// TIA Portal V17 export
// export: Created 2025-03-10T12:16:33.8598493Z, ExportSetting WithDefaults, DisplayName Totally Integrated Automation Portal, DisplayVersion V17 Update 8, DisplayName TIA Portal Openness, DisplayVersion V17 Update 8, DisplayName TIA Portal Version Control Interface, DisplayVersion V17, DisplayName SINAMICS Startdrive Advanced, DisplayVersion V17 SP2, DisplayName SINAMICS Startdrive G110M, G120, G120C, G120D, G120P, G115D, DisplayVersion V17 SP2, DisplayName SINAMICS Startdrive G130, G150, S120, S150, SINAMICS MV, S210, DisplayVersion V17 SP2, DisplayName STEP 7 Professional, DisplayVersion V17 Update 8, DisplayName SINUMERIK ONE STEP 7 Toolbox, DisplayVersion V17 Update 12, DisplayName SINUMERIK 840D sl STEP 7 Toolbox, DisplayVersion V17 Update 12, DisplayName STEP 7 Safety, DisplayVersion V17 Update 6, DisplayName WinCC Advanced, DisplayVersion V17 Update 8
FUNCTION_BLOCK "FB1452_AUXILIARY_COOLING_SYSTEM"   // FB1452, LAD
{ S7_Optimized_Access := 'FALSE' }
AUTHOR : ETXETAR
VERSION : 1.0
// stored: AutoNumber false, IsIECCheckEnabled false, SetENOAutomatically false, UDAEnableTagReadback false
   VAR_INPUT
      OPTIONS_0 : Byte := 2#0000_0000;   // OPTIONS 0
      OPTIONS_1 : Byte := 2#0000_0000;   // OPTIONS 1
      CIRCUIT_BREAKER_INPUT : Bool;   // CIRCUIT BREAKER INPUT
      CONTACTOR_FEEDBACK : Bool;   // CONTACTOR FEEDBACK INPUT
      LOW_LEVEL_ALM : Bool;   // UNIT 01 LOW LEVEL ALARM
      OVERTEMPERATURE_ALM : Bool;   // UNIT 01 OVERTEMPERATURE ALARM
      U01_FLOW_ACTUAL_RAW_VALUE : Int;   // UNIT 01 FLOW ACTUAL RAW VALUE
      U01_TEMP_ACTUAL_RAW_VALUE : Int;   // UNIT 01 TEMPURATURE ACTUAL RAW VALUE
      U02_FLOW_ACTUAL_RAW_VALUE : Int;   // UNIT 02 FLOW ACTUAL RAW VALUE
      U02_TEMP_ACTUAL_RAW_VALUE : Int;   // UNIT 02 TEMPURATURE ACTUAL RAW VALUE
      HMI_REQ_LINE : Bool;   // HMI REQUEST LINE
   END_VAR
   VAR_OUTPUT
      U01_U02_BREAKER_TRIPPED_ALARM : Bool;   // UNIT 01 & UNIT 02 CIRCUIT BREAKER TRIPPED ALARM
      U01_U02_CONTACTOR_FEEDBACK_ALARM : Bool;   // UNIT 01 & UNIT 02 CONTACTOR FEEDBACK ALARM
      U01_U02_LOW_LEVEL_INPUT_ALARM : Bool;   // UNIT 01 & UNIT 02 LOW LEVEL INPUT ALARM
      U01_U02_OVERTEMPERATURE_INPUT_ALARM : Bool;   // UNIT 01 & UNIT 02 OVERTEMPERATURE INPUT ALARM
      U01_FLOW_FEEDBACK_ALARM : Bool;   // UNIT 01 FLOW FEEDBACK ALARM
      U01_FLOW_HIGH_LIMIT_ALARM : Bool;   // UNIT 01 FLOW HIGH LIMIT ALARM
      U01_FLOW_HIGH_LIMIT_WARNING : Bool;   // UNIT 01 FLOW HIGH LIMIT WARNING
      U01_FLOW_LOW_LIMIT_ALARM : Bool;   // UNIT 01 FLOW LOW LIMIT ALARM
      U01_FLOW_LOW_LIMIT_WARNING : Bool;   // UNIT 01 FLOW LOW LIMIT WARNING
      U01_TEMP_HIGH_LIMIT_ALARM : Bool;   // UNIT 01 TEMPERATURE HIGH LIMIT ALARM
      U01_TEMP_HIGH_LIMIT_WARNING : Bool;   // UNIT 01 TEMPERATURE HIGH LIMIT WARNING
      U01_TEMP_LOW_LIMIT_ALARM : Bool;   // UNIT 01 TEMPERATURE LOW LIMIT ALARM
      U01_TEMP_LOW_LIMIT_WARNING : Bool;   // UNIT 01 TEMPERATURE LOW LIMIT WARNING
      U01_FLOW_SETPOINT_ALARM : Bool;   // UNIT 01 FLOW SETPOINT ALARM
      U01_TEMP_SETPOINT_ALARM : Bool;   // UNIT 01 TEMPERATURE SETPOINT ALARM
      U02_FLOW_FEEDBACK_ALARM : Bool;   // UNIT 02 FLOW FEEDBACK ALARM
      U02_FLOW_HIGH_LIMIT_ALARM : Bool;   // UNIT 01 FLOW HIGH LIMIT ALARM
      U02_FLOW_HIGH_LIMIT_WARNING : Bool;   // UNIT 01 FLOW HIGH LIMIT WARNING
      U02_FLOW_LOW_LIMIT_ALARM : Bool;   // UNIT 01 FLOW LOW LIMIT ALARM
      U02_FLOW_LOW_LIMIT_WARNING : Bool;   // UNIT 01 FLOW LOW LIMIT WARNING
      U02_TEMP_HIGH_LIMIT_ALARM : Bool;   // UNIT 01 TEMPERATURE HIGH LIMIT ALARM
      U02_TEMP_HIGH_LIMIT_WARNING : Bool;   // UNIT 01 TEMPERATURE HIGH LIMIT WARNING
      U02_TEMP_LOW_LIMIT_ALARM : Bool;   // UNIT 01 TEMPERATURE LOW LIMIT ALARM
      U02_TEMP_LOW_LIMIT_WARNING : Bool;   // UNIT 01 TEMPERATURE LOW LIMIT WARNING
      U02_FLOW_SETPOINT_ALARM : Bool;   // UNIT 01 FLOW SETPOINT ALARM
      U02_TEMP_SETPOINT_ALARM : Bool;   // UNIT 01 TEMPERATURE SETPOINT ALARM
      HMI_POWER_UP_COND_OFF : Bool;   // HMI POWER UP CONDITIONS OFF
      HMI_POWER_UP_COND_ON : Bool;   // HMI POWER UP CONDITIONS ON
      HMI_POWER_UP_EXECU_LEFT : Bool;   // HMI POWER UP EXECUTABLE LEFT
      HMI_POWER_UP_EXECU_RIGHT : Bool;   // HMI POWER UP EXECUTABLE RIGHT
      MAIN_VALVE : Bool;   // MAIN VALVE OUTPUT
   END_VAR
   VAR DB_SPECIFIC
      SWITCH_ON_GENERAL_CONDITIONS : Bool;   // SWITCH ON GENERAL CONDITIONS
      SWITCH_ON_INITIAL_CONDITIONS : Bool;   // SWITCH ON INITIAL CONDITIONS
      SWITCH_ON_MANUAL_REQUEST : Bool;   // SWITCH ON MANUAL REQUEST
      SWITCH_ON_AUTO_REQUEST : Bool;   // SWITCH ON AUTO REQUEST
      SWITCH_ON_GLOBAL_REQUEST : Bool;   // SWITCH ON GLOBAL REQUEST
      SWITCH_ON_COMMAND : Bool;   // SWITCH ON COMMAND
      SWITCH_ON : Bool;   // SWITCH ON
      IN_SERVICE : Bool;   // IN SERVICE
      SWITCH_OFF_GENERAL_CONDITIONS : Bool;   // SWITCH OFF GENERAL CONDITIONS
      SWITCH_OFF_INITIAL_CONDITIONS : Bool;   // SWITCH OFF INITIAL CONDITIONS
      SWITCH_OFF_MANUAL_REQUEST : Bool;   // SWITCH OFF MANUAL REQUEST
      SWITCH_OFF_AUTO_REQUEST : Bool;   // SWITCH OFF AUTO REQUEST
      SWITCH_OFF_GLOBAL_REQUEST : Bool;   // SWITCH OFF GLOBAL REQUEST
      SWITCH_OFF_COMMAND : Bool;   // SWITCH OFF COMMAND
      SWITCH_OFF : Bool;   // SWITCH OFF
      OUT_OF_SERVICE : Bool;   // OUT OF SERVICE
      MANUAL_REQUEST_HELP : Bool;   // MANUAL REQUEST HELP
      SWITCH_ON_GENERAL_CONDITION_HELP : Bool;   // SWITCH ON GENERAL CONDITION HELP
      SWITCH_ON_INITIAL_CONDITION_HELP : Bool;   // SWITCH ON INITIAL CONDITION HELP
      SWITCH_OFF_GENERAL_CONDITION_HELP : Bool;   // SWITCH OFF GENERAL CONDITION HELP
      SWITCH_OFF_INITIAL_CONDITION_HELP : Bool;   // SWITCH OFF INITIAL CONDITION HELP
      ANY_ACTIVE_ALARM : Bool;   // ANY ACTIVE ALARM
      SEOC_ALARMS : Bool;   // STOP END OF CYCLE ALARMS
      WARNINGS : Bool;   // WARNINGS
      WARNINGS_GONE : Bool;   // WARNINGS GONE
      UNIT_01_FLOW_FEEDBACK_INPUT : Bool;   // UNIT 01 FLOW PRESENT INPUT
      UNIT_02_FLOW_FEEDBACK_INPUT : Bool;   // UNIT 02 FLOW PRESENT INPUT
      TOTAL_FLOW_FEEDBACK_INPUT : Bool;   // TOTAL FLOW PRESENT INPUT
      AUX_COOLING_SENSOR_U01_VALUES { ExternalAccessible := 'False'; ExternalVisible := 'False'; ExternalWritable := 'False'} : "COOLING_SENSOR";
      AUX_COOLING_SENSOR_U02_VALUES { ExternalAccessible := 'False'; ExternalVisible := 'False'; ExternalWritable := 'False'} : "COOLING_SENSOR";
      TIMER_CONVEYOR_CONTACTOR_RELAY_ALARM : TON_TIME;   // PRESSURE TIMER
   END_VAR
   VAR_TEMP
      INPUTS_MASK : Byte;   // INPUT MASK
      O_BYTE_0 : Struct   // OPTIONS BYTE 0
         GEN_CIRCUIT_BREAKER : Bool;   // GENERAL CIRCUIT BREAKER OPTION
         GEN_CONTACTOR_FEEDBACK : Bool;   // GENERAL CONTACTOR FEEDBACK OPTION
         U01_FLOW_SETPOINT_ALARM : Bool;   // UNIT 01 FLOW SETPOINT ALARM
         U01_TEMP_SETPOINT_ALARM : Bool;   // UNIT 01 TEMPERATURE SETPOINT ALARM
         SPARE_2 : Bool;
         SPARE_3 : Bool;
         SPARE_4 : Bool;
         SPARE_5 : Bool;
      END_STRUCT;
      O_BYTE_1 : Struct   // OPTIONS BYTE 1
         FIRST_FEEDBACK_FLOW_TEMP_SENSOR : Bool;   // FIRST FEEDBACK FLOW TEMP SENSOR
         SECOND_FEEDBACK_FLOW_TEMP_SENSOR : Bool;   // SECOND FEEDBACK FLOW TEMP SENSOR
         U02_FLOW_SETPOINT_ALARM : Bool;   // UNIT 02 FLOW SETPOINT ALARM
         U02_TEMP_SETPOINT_ALARM : Bool;   // UNIT 02 TEMPERATURE SETPOINT ALARM
         SPARE_2 : Bool;
         SPARE_3 : Bool;
         SPARE_4 : Bool;
         SPARE_5 : Bool;
      END_STRUCT;
      DB_NUMBER : DInt;   // DB NUMBER FOR ALARM DECODING
      FLOW_AUX : Real;
      TEMPERATURE_AUX : Int;
   END_VAR
   // TIMER_CONVEYOR_CONTACTOR_RELAY_ALARM.PT := T#1M;
   VAR_TEMP   // added for the SCL form of the ladder/FBD networks
      _w1 : Bool;
   END_VAR
BEGIN

NETWORK
TITLE = READ INSTANCE DB
      L     DINO;
      +     10#800000;
      T     #DB_NUMBER;


REGION Network 2: OPTIONS
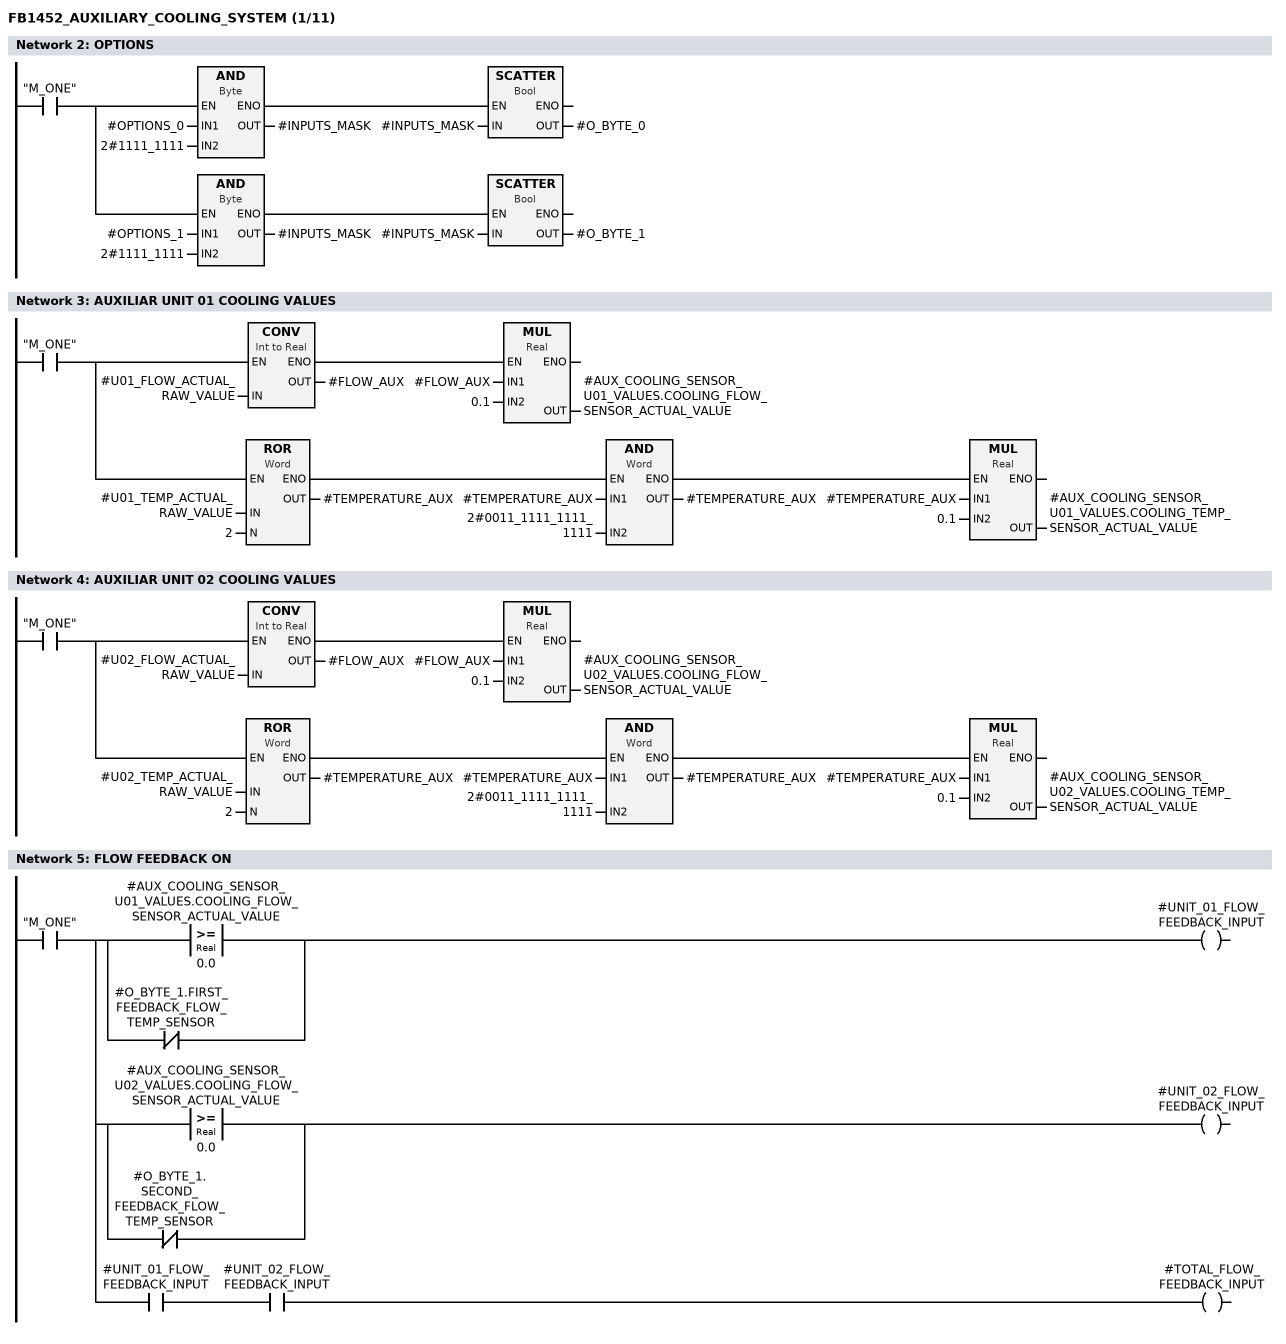
   RUNG wire#powerrail
      Contact( "M_ONE" )
      wire#w1
      { S7_Templates := "SrcType := Byte"; S7_GenerateENO := "TRUE" } And(in1 := #OPTIONS_0, in2 := 2#1111_1111, out => #INPUTS_MASK)
      { S7_Templates := "[dest_type := Bool, src_type := Byte]" } SCATTER(IN := #INPUTS_MASK, OUT => #O_BYTE_0)
   END_RUNG
   RUNG wire#w1
      { S7_Templates := "SrcType := Byte"; S7_GenerateENO := "TRUE" } And(in1 := #OPTIONS_1, in2 := 2#1111_1111, out => #INPUTS_MASK)
      { S7_Templates := "[dest_type := Bool, src_type := Byte]" } SCATTER(IN := #INPUTS_MASK, OUT => #O_BYTE_1)
   END_RUNG
   // the same network as SCL:
   IF "M_ONE" THEN #INPUTS_MASK := #OPTIONS_0 AND 2#1111_1111; END_IF;
   #_w1 := "M_ONE";
   IF #_w1 THEN
       SCATTER(IN := #INPUTS_MASK, OUT => #O_BYTE_0);
       #INPUTS_MASK := #OPTIONS_1 AND 2#1111_1111;
       SCATTER(IN := #INPUTS_MASK, OUT => #O_BYTE_1);
   END_IF;
END_REGION

REGION Network 3: AUXILIAR UNIT 01 COOLING VALUES
   IF "M_ONE" THEN
       #FLOW_AUX := INT_TO_REAL(#U01_FLOW_ACTUAL_RAW_VALUE);
       #AUX_COOLING_SENSOR_U01_VALUES.COOLING_FLOW_SENSOR_ACTUAL_VALUE := #FLOW_AUX * 0.1;
       #TEMPERATURE_AUX := ROR(IN := #U01_TEMP_ACTUAL_RAW_VALUE, N := 2);
       #TEMPERATURE_AUX := #TEMPERATURE_AUX AND 2#0011_1111_1111_1111;
       #AUX_COOLING_SENSOR_U01_VALUES.COOLING_TEMP_SENSOR_ACTUAL_VALUE := #TEMPERATURE_AUX * 0.1;
   END_IF;
END_REGION

REGION Network 4: AUXILIAR UNIT 02 COOLING VALUES
   IF "M_ONE" THEN
       #FLOW_AUX := INT_TO_REAL(#U02_FLOW_ACTUAL_RAW_VALUE);
       #AUX_COOLING_SENSOR_U02_VALUES.COOLING_FLOW_SENSOR_ACTUAL_VALUE := #FLOW_AUX * 0.1;
       #TEMPERATURE_AUX := ROR(IN := #U02_TEMP_ACTUAL_RAW_VALUE, N := 2);
       #TEMPERATURE_AUX := #TEMPERATURE_AUX AND 2#0011_1111_1111_1111;
       #AUX_COOLING_SENSOR_U02_VALUES.COOLING_TEMP_SENSOR_ACTUAL_VALUE := #TEMPERATURE_AUX * 0.1;
   END_IF;
END_REGION

REGION Network 5: FLOW FEEDBACK ON
   RUNG wire#powerrail
      Contact( "M_ONE" )
      wire#w1
      { S7_Templates := "SrcType := Real" } GE_Contact(in1 := #AUX_COOLING_SENSOR_U01_VALUES.COOLING_FLOW_SENSOR_ACTUAL_VALUE, in2 := 0.0)
      wire#w2
      Coil( #UNIT_01_FLOW_FEEDBACK_INPUT )
   END_RUNG
   RUNG wire#w1
      I_Contact( #O_BYTE_1.FIRST_FEEDBACK_FLOW_TEMP_SENSOR )
   END_RUNG wire#w2
   RUNG wire#w1
      { S7_Templates := "SrcType := Real" } GE_Contact(in1 := #AUX_COOLING_SENSOR_U02_VALUES.COOLING_FLOW_SENSOR_ACTUAL_VALUE, in2 := 0.0)
      wire#w3
      Coil( #UNIT_02_FLOW_FEEDBACK_INPUT )
   END_RUNG
   RUNG wire#w1
      I_Contact( #O_BYTE_1.SECOND_FEEDBACK_FLOW_TEMP_SENSOR )
   END_RUNG wire#w3
   RUNG wire#w1
      Contact( #UNIT_01_FLOW_FEEDBACK_INPUT )
      Contact( #UNIT_02_FLOW_FEEDBACK_INPUT )
      Coil( #TOTAL_FLOW_FEEDBACK_INPUT )
   END_RUNG
   // the same network as SCL:
   #UNIT_01_FLOW_FEEDBACK_INPUT := "M_ONE" AND ((#AUX_COOLING_SENSOR_U01_VALUES.COOLING_FLOW_SENSOR_ACTUAL_VALUE >= 0.0) OR NOT #O_BYTE_1.FIRST_FEEDBACK_FLOW_TEMP_SENSOR);
   #UNIT_02_FLOW_FEEDBACK_INPUT := "M_ONE" AND ((#AUX_COOLING_SENSOR_U02_VALUES.COOLING_FLOW_SENSOR_ACTUAL_VALUE >= 0.0) OR NOT #O_BYTE_1.SECOND_FEEDBACK_FLOW_TEMP_SENSOR);
   #TOTAL_FLOW_FEEDBACK_INPUT := "M_ONE" AND #UNIT_01_FLOW_FEEDBACK_INPUT AND #UNIT_02_FLOW_FEEDBACK_INPUT;
END_REGION

REGION Network 6: SWITCH ON GENERAL CONDITIONS
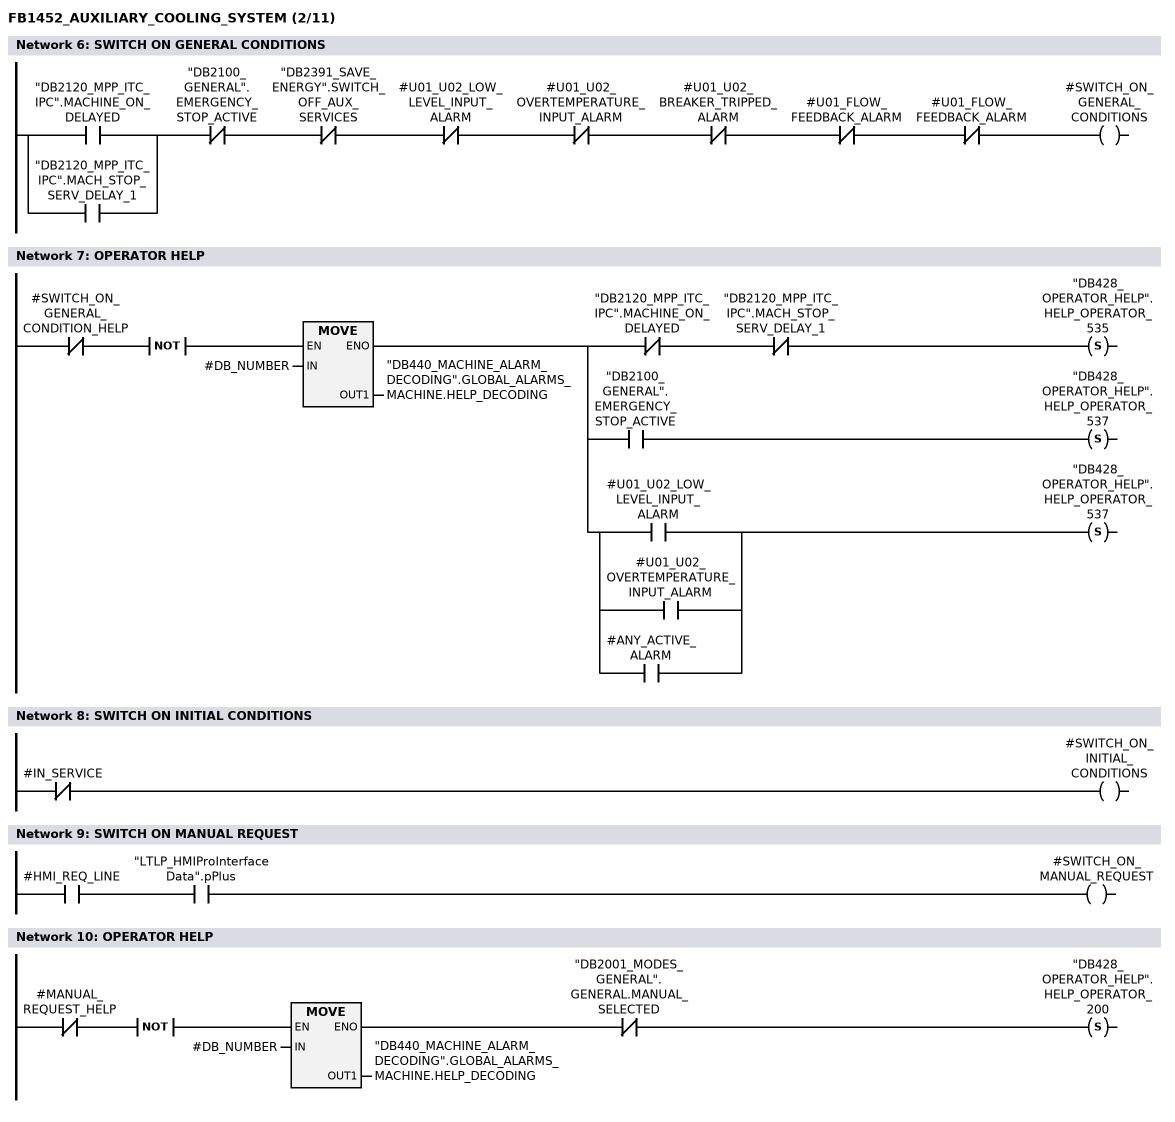
   RUNG wire#powerrail
      Contact( "DB2120_MPP_ITC_IPC".MACHINE_ON_DELAYED )
      wire#w1
      I_Contact( "DB2100_GENERAL".EMERGENCY_STOP_ACTIVE )
      I_Contact( "DB2391_SAVE_ENERGY".SWITCH_OFF_AUX_SERVICES )
      I_Contact( #U01_U02_LOW_LEVEL_INPUT_ALARM )
      I_Contact( #U01_U02_OVERTEMPERATURE_INPUT_ALARM )
      I_Contact( #U01_U02_BREAKER_TRIPPED_ALARM )
      I_Contact( #U01_FLOW_FEEDBACK_ALARM )
      I_Contact( #U01_FLOW_FEEDBACK_ALARM )
      Coil( #SWITCH_ON_GENERAL_CONDITIONS )
   END_RUNG
   RUNG wire#powerrail
      Contact( "DB2120_MPP_ITC_IPC".MACH_STOP_SERV_DELAY_1 )
   END_RUNG wire#w1
   // the same network as SCL:
   #SWITCH_ON_GENERAL_CONDITIONS := ("DB2120_MPP_ITC_IPC".MACHINE_ON_DELAYED OR "DB2120_MPP_ITC_IPC".MACH_STOP_SERV_DELAY_1) AND NOT "DB2100_GENERAL".EMERGENCY_STOP_ACTIVE AND NOT "DB2391_SAVE_ENERGY".SWITCH_OFF_AUX_SERVICES AND NOT #U01_U02_LOW_LEVEL_INPUT_ALARM AND NOT #U01_U02_OVERTEMPERATURE_INPUT_ALARM AND NOT #U01_U02_BREAKER_TRIPPED_ALARM AND NOT #U01_FLOW_FEEDBACK_ALARM AND NOT #U01_FLOW_FEEDBACK_ALARM;
END_REGION

REGION Network 7: OPERATOR HELP
   RUNG wire#powerrail
      I_Contact( #SWITCH_ON_GENERAL_CONDITION_HELP )
      Not()
      { S7_GenerateENO := "TRUE" } Move(in := #DB_NUMBER, out1 => "DB440_MACHINE_ALARM_DECODING".GLOBAL_ALARMS_MACHINE.HELP_DECODING)
      wire#w1
      I_Contact( "DB2120_MPP_ITC_IPC".MACHINE_ON_DELAYED )
      I_Contact( "DB2120_MPP_ITC_IPC".MACH_STOP_SERV_DELAY_1 )
      S_Coil( "DB428_OPERATOR_HELP".HELP_OPERATOR_535 )
   END_RUNG
   RUNG wire#w1
      Contact( "DB2100_GENERAL".EMERGENCY_STOP_ACTIVE )
      S_Coil( "DB428_OPERATOR_HELP".HELP_OPERATOR_537 )
   END_RUNG
   RUNG wire#w1
      Contact( #U01_U02_LOW_LEVEL_INPUT_ALARM )
      wire#w2
      S_Coil( "DB428_OPERATOR_HELP".HELP_OPERATOR_537 )
   END_RUNG
   RUNG wire#w1
      Contact( #U01_U02_OVERTEMPERATURE_INPUT_ALARM )
   END_RUNG wire#w2
   RUNG wire#w1
      Contact( #ANY_ACTIVE_ALARM )
   END_RUNG wire#w2
   // the same network as SCL:
   // ENO of a box is taken as its EN; it also drops when the box reports an error
   #_w1 := NOT (NOT #SWITCH_ON_GENERAL_CONDITION_HELP);
   IF #_w1 THEN "DB440_MACHINE_ALARM_DECODING".GLOBAL_ALARMS_MACHINE.HELP_DECODING := #DB_NUMBER; END_IF;
   IF #_w1 AND NOT "DB2120_MPP_ITC_IPC".MACHINE_ON_DELAYED AND NOT "DB2120_MPP_ITC_IPC".MACH_STOP_SERV_DELAY_1 THEN
       "DB428_OPERATOR_HELP".HELP_OPERATOR_535 := TRUE;
   END_IF;
   IF #_w1 AND "DB2100_GENERAL".EMERGENCY_STOP_ACTIVE THEN
       "DB428_OPERATOR_HELP".HELP_OPERATOR_537 := TRUE;
   END_IF;
   IF #_w1 AND (#U01_U02_LOW_LEVEL_INPUT_ALARM OR #U01_U02_OVERTEMPERATURE_INPUT_ALARM OR #ANY_ACTIVE_ALARM) THEN
       "DB428_OPERATOR_HELP".HELP_OPERATOR_537 := TRUE;
   END_IF;
END_REGION

REGION Network 8: SWITCH ON INITIAL CONDITIONS
   RUNG wire#powerrail
      I_Contact( #IN_SERVICE )
      Coil( #SWITCH_ON_INITIAL_CONDITIONS )
   END_RUNG
   // the same network as SCL:
   #SWITCH_ON_INITIAL_CONDITIONS := NOT #IN_SERVICE;
END_REGION

REGION Network 9: SWITCH ON MANUAL REQUEST
   RUNG wire#powerrail
      Contact( #HMI_REQ_LINE )
      Contact( "LTLP_HMIProInterfaceData".pPlus )
      Coil( #SWITCH_ON_MANUAL_REQUEST )
   END_RUNG
   // the same network as SCL:
   #SWITCH_ON_MANUAL_REQUEST := #HMI_REQ_LINE AND "LTLP_HMIProInterfaceData".pPlus;
END_REGION

REGION Network 10: OPERATOR HELP
   RUNG wire#powerrail
      I_Contact( #MANUAL_REQUEST_HELP )
      Not()
      { S7_GenerateENO := "TRUE" } Move(in := #DB_NUMBER, out1 => "DB440_MACHINE_ALARM_DECODING".GLOBAL_ALARMS_MACHINE.HELP_DECODING)
      I_Contact( "DB2001_MODES_GENERAL".GENERAL.MANUAL_SELECTED )
      S_Coil( "DB428_OPERATOR_HELP".HELP_OPERATOR_200 )
   END_RUNG
   // the same network as SCL:
   // ENO of a box is taken as its EN; it also drops when the box reports an error
   #_w1 := NOT (NOT #MANUAL_REQUEST_HELP);
   IF #_w1 THEN "DB440_MACHINE_ALARM_DECODING".GLOBAL_ALARMS_MACHINE.HELP_DECODING := #DB_NUMBER; END_IF;
   IF #_w1 AND NOT "DB2001_MODES_GENERAL".GENERAL.MANUAL_SELECTED THEN
       "DB428_OPERATOR_HELP".HELP_OPERATOR_200 := TRUE;
   END_IF;
END_REGION

REGION Network 11: SWITCH ON AUTO REQUEST
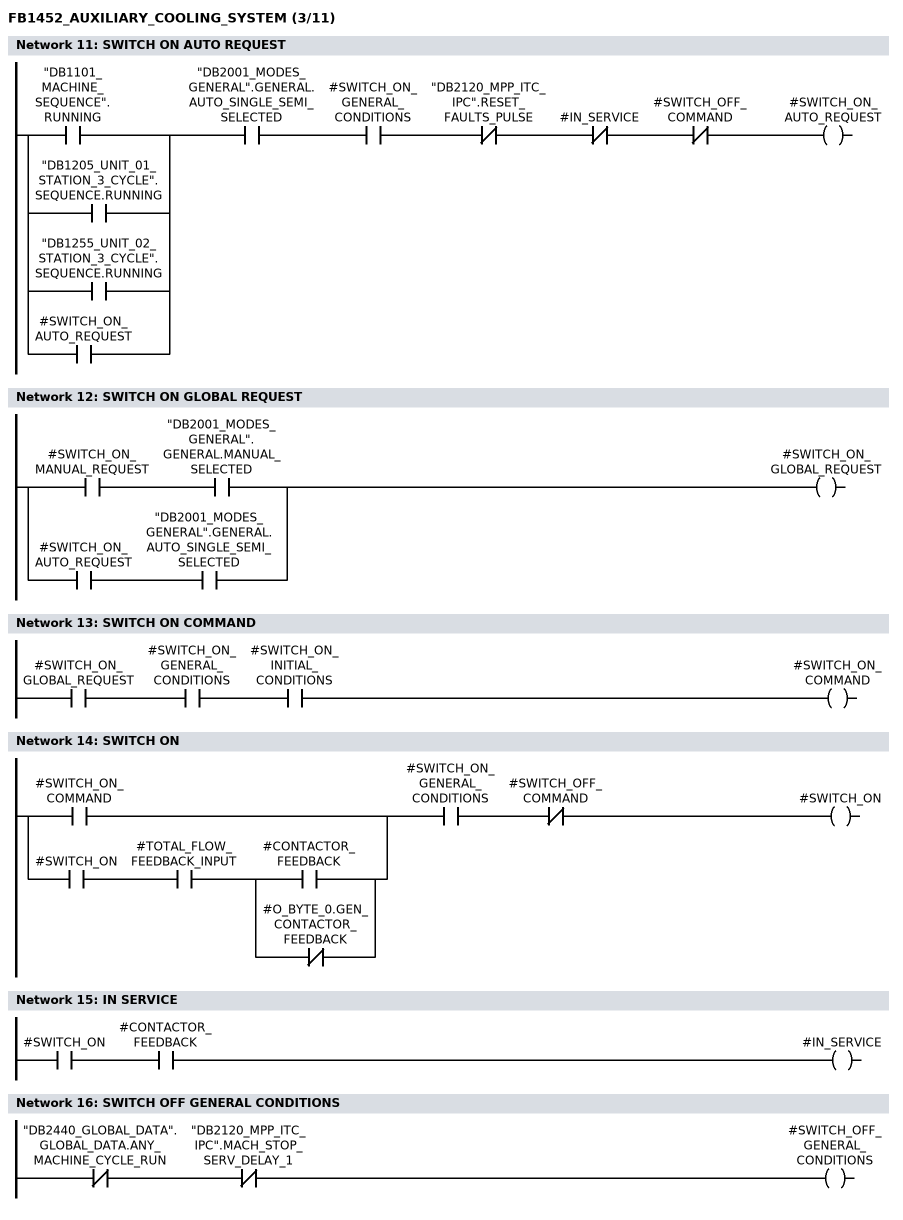
   RUNG wire#powerrail
      Contact( "DB1101_MACHINE_SEQUENCE".RUNNING )
      wire#w1
      Contact( "DB2001_MODES_GENERAL".GENERAL.AUTO_SINGLE_SEMI_SELECTED )
      Contact( #SWITCH_ON_GENERAL_CONDITIONS )
      I_Contact( "DB2120_MPP_ITC_IPC".RESET_FAULTS_PULSE )
      I_Contact( #IN_SERVICE )
      I_Contact( #SWITCH_OFF_COMMAND )
      Coil( #SWITCH_ON_AUTO_REQUEST )
   END_RUNG
   RUNG wire#powerrail
      Contact( "DB1205_UNIT_01_STATION_3_CYCLE".SEQUENCE.RUNNING )
   END_RUNG wire#w1
   RUNG wire#powerrail
      Contact( "DB1255_UNIT_02_STATION_3_CYCLE".SEQUENCE.RUNNING )
   END_RUNG wire#w1
   RUNG wire#powerrail
      Contact( #SWITCH_ON_AUTO_REQUEST )
   END_RUNG wire#w1
   // the same network as SCL:
   #SWITCH_ON_AUTO_REQUEST := ("DB1101_MACHINE_SEQUENCE".RUNNING OR "DB1205_UNIT_01_STATION_3_CYCLE".SEQUENCE.RUNNING OR "DB1255_UNIT_02_STATION_3_CYCLE".SEQUENCE.RUNNING OR #SWITCH_ON_AUTO_REQUEST) AND "DB2001_MODES_GENERAL".GENERAL.AUTO_SINGLE_SEMI_SELECTED AND #SWITCH_ON_GENERAL_CONDITIONS AND NOT "DB2120_MPP_ITC_IPC".RESET_FAULTS_PULSE AND NOT #IN_SERVICE AND NOT #SWITCH_OFF_COMMAND;
END_REGION

REGION Network 12: SWITCH ON GLOBAL REQUEST
   RUNG wire#powerrail
      Contact( #SWITCH_ON_MANUAL_REQUEST )
      Contact( "DB2001_MODES_GENERAL".GENERAL.MANUAL_SELECTED )
      wire#w1
      Coil( #SWITCH_ON_GLOBAL_REQUEST )
   END_RUNG
   RUNG wire#powerrail
      Contact( #SWITCH_ON_AUTO_REQUEST )
      Contact( "DB2001_MODES_GENERAL".GENERAL.AUTO_SINGLE_SEMI_SELECTED )
   END_RUNG wire#w1
   // the same network as SCL:
   #SWITCH_ON_GLOBAL_REQUEST := (#SWITCH_ON_MANUAL_REQUEST AND "DB2001_MODES_GENERAL".GENERAL.MANUAL_SELECTED) OR (#SWITCH_ON_AUTO_REQUEST AND "DB2001_MODES_GENERAL".GENERAL.AUTO_SINGLE_SEMI_SELECTED);
END_REGION

REGION Network 13: SWITCH ON COMMAND
   RUNG wire#powerrail
      Contact( #SWITCH_ON_GLOBAL_REQUEST )
      Contact( #SWITCH_ON_GENERAL_CONDITIONS )
      Contact( #SWITCH_ON_INITIAL_CONDITIONS )
      Coil( #SWITCH_ON_COMMAND )
   END_RUNG
   // the same network as SCL:
   #SWITCH_ON_COMMAND := #SWITCH_ON_GLOBAL_REQUEST AND #SWITCH_ON_GENERAL_CONDITIONS AND #SWITCH_ON_INITIAL_CONDITIONS;
END_REGION

REGION Network 14: SWITCH ON
   RUNG wire#powerrail
      Contact( #SWITCH_ON_COMMAND )
      wire#w1
      Contact( #SWITCH_ON_GENERAL_CONDITIONS )
      I_Contact( #SWITCH_OFF_COMMAND )
      Coil( #SWITCH_ON )
   END_RUNG
   RUNG wire#powerrail
      Contact( #SWITCH_ON )
      Contact( #TOTAL_FLOW_FEEDBACK_INPUT )
      wire#w2
      Contact( #CONTACTOR_FEEDBACK )
   END_RUNG wire#w1
   RUNG wire#w2
      I_Contact( #O_BYTE_0.GEN_CONTACTOR_FEEDBACK )
   END_RUNG wire#w1
   // the same network as SCL:
   #SWITCH_ON := (#SWITCH_ON_COMMAND OR (#SWITCH_ON AND #TOTAL_FLOW_FEEDBACK_INPUT AND (#CONTACTOR_FEEDBACK OR NOT #O_BYTE_0.GEN_CONTACTOR_FEEDBACK))) AND #SWITCH_ON_GENERAL_CONDITIONS AND NOT #SWITCH_OFF_COMMAND;
END_REGION

REGION Network 15: IN SERVICE
   RUNG wire#powerrail
      Contact( #SWITCH_ON )
      Contact( #CONTACTOR_FEEDBACK )
      Coil( #IN_SERVICE )
   END_RUNG
   // the same network as SCL:
   #IN_SERVICE := #SWITCH_ON AND #CONTACTOR_FEEDBACK;
END_REGION

REGION Network 16: SWITCH OFF GENERAL CONDITIONS
   RUNG wire#powerrail
      I_Contact( "DB2440_GLOBAL_DATA".GLOBAL_DATA.ANY_MACHINE_CYCLE_RUN )
      I_Contact( "DB2120_MPP_ITC_IPC".MACH_STOP_SERV_DELAY_1 )
      Coil( #SWITCH_OFF_GENERAL_CONDITIONS )
   END_RUNG
   // the same network as SCL:
   #SWITCH_OFF_GENERAL_CONDITIONS := NOT "DB2440_GLOBAL_DATA".GLOBAL_DATA.ANY_MACHINE_CYCLE_RUN AND NOT "DB2120_MPP_ITC_IPC".MACH_STOP_SERV_DELAY_1;
END_REGION

REGION Network 17: OPERATOR HELP
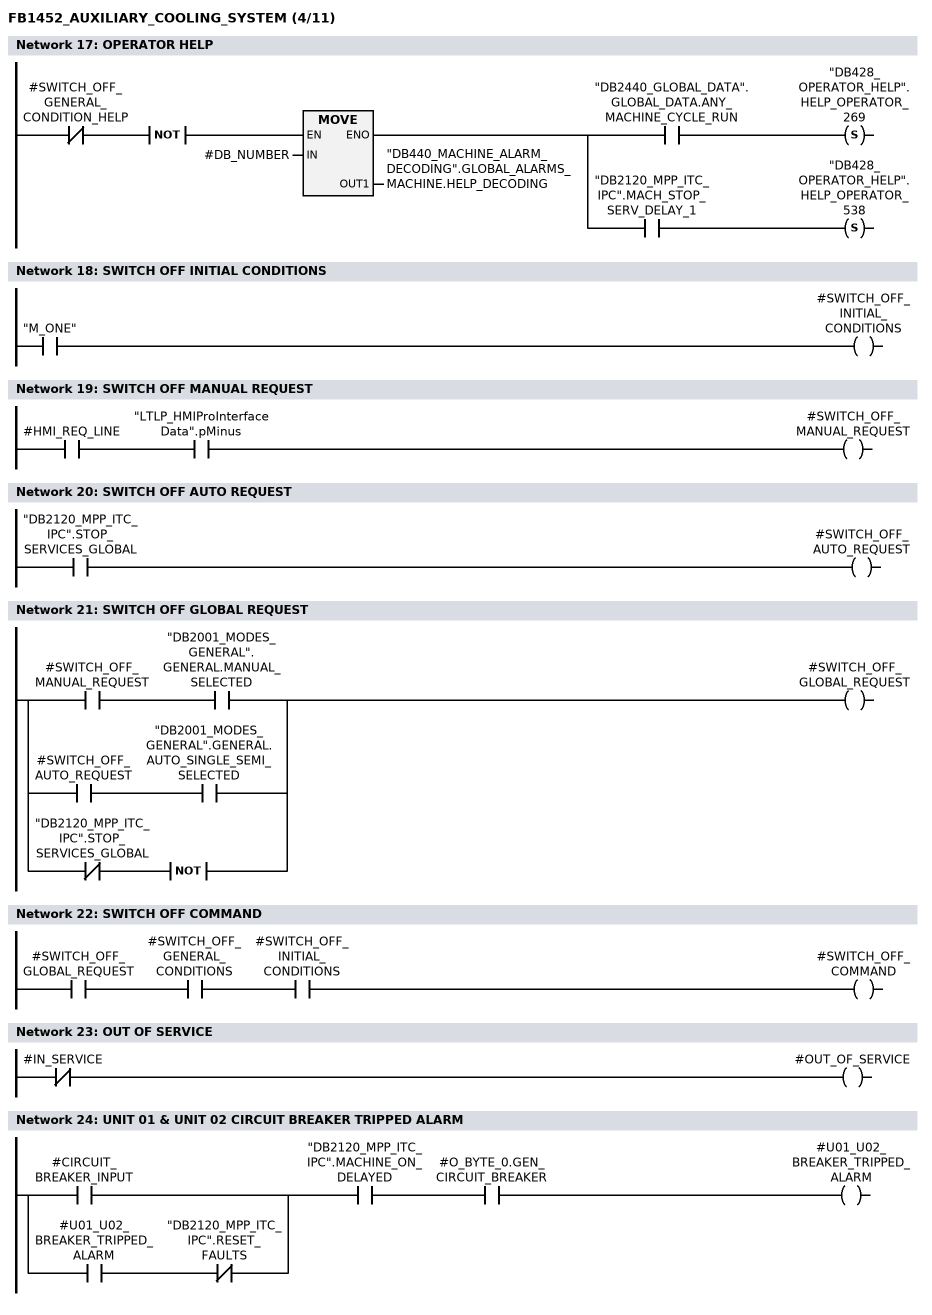
   RUNG wire#powerrail
      I_Contact( #SWITCH_OFF_GENERAL_CONDITION_HELP )
      Not()
      { S7_GenerateENO := "TRUE" } Move(in := #DB_NUMBER, out1 => "DB440_MACHINE_ALARM_DECODING".GLOBAL_ALARMS_MACHINE.HELP_DECODING)
      wire#w1
      Contact( "DB2440_GLOBAL_DATA".GLOBAL_DATA.ANY_MACHINE_CYCLE_RUN )
      S_Coil( "DB428_OPERATOR_HELP".HELP_OPERATOR_269 )
   END_RUNG
   RUNG wire#w1
      Contact( "DB2120_MPP_ITC_IPC".MACH_STOP_SERV_DELAY_1 )
      S_Coil( "DB428_OPERATOR_HELP".HELP_OPERATOR_538 )
   END_RUNG
   // the same network as SCL:
   // ENO of a box is taken as its EN; it also drops when the box reports an error
   #_w1 := NOT (NOT #SWITCH_OFF_GENERAL_CONDITION_HELP);
   IF #_w1 THEN "DB440_MACHINE_ALARM_DECODING".GLOBAL_ALARMS_MACHINE.HELP_DECODING := #DB_NUMBER; END_IF;
   IF #_w1 AND "DB2440_GLOBAL_DATA".GLOBAL_DATA.ANY_MACHINE_CYCLE_RUN THEN
       "DB428_OPERATOR_HELP".HELP_OPERATOR_269 := TRUE;
   END_IF;
   IF #_w1 AND "DB2120_MPP_ITC_IPC".MACH_STOP_SERV_DELAY_1 THEN
       "DB428_OPERATOR_HELP".HELP_OPERATOR_538 := TRUE;
   END_IF;
END_REGION

REGION Network 18: SWITCH OFF INITIAL CONDITIONS
   RUNG wire#powerrail
      Contact( "M_ONE" )
      Coil( #SWITCH_OFF_INITIAL_CONDITIONS )
   END_RUNG
   // the same network as SCL:
   #SWITCH_OFF_INITIAL_CONDITIONS := "M_ONE";
END_REGION

REGION Network 19: SWITCH OFF MANUAL REQUEST
   RUNG wire#powerrail
      Contact( #HMI_REQ_LINE )
      Contact( "LTLP_HMIProInterfaceData".pMinus )
      Coil( #SWITCH_OFF_MANUAL_REQUEST )
   END_RUNG
   // the same network as SCL:
   #SWITCH_OFF_MANUAL_REQUEST := #HMI_REQ_LINE AND "LTLP_HMIProInterfaceData".pMinus;
END_REGION

REGION Network 20: SWITCH OFF AUTO REQUEST
   RUNG wire#powerrail
      Contact( "DB2120_MPP_ITC_IPC".STOP_SERVICES_GLOBAL )
      Coil( #SWITCH_OFF_AUTO_REQUEST )
   END_RUNG
   // the same network as SCL:
   #SWITCH_OFF_AUTO_REQUEST := "DB2120_MPP_ITC_IPC".STOP_SERVICES_GLOBAL;
END_REGION

REGION Network 21: SWITCH OFF GLOBAL REQUEST
   RUNG wire#powerrail
      Contact( #SWITCH_OFF_MANUAL_REQUEST )
      Contact( "DB2001_MODES_GENERAL".GENERAL.MANUAL_SELECTED )
      wire#w1
      Coil( #SWITCH_OFF_GLOBAL_REQUEST )
   END_RUNG
   RUNG wire#powerrail
      Contact( #SWITCH_OFF_AUTO_REQUEST )
      Contact( "DB2001_MODES_GENERAL".GENERAL.AUTO_SINGLE_SEMI_SELECTED )
   END_RUNG wire#w1
   RUNG wire#powerrail
      I_Contact( "DB2120_MPP_ITC_IPC".STOP_SERVICES_GLOBAL )
      Not()
   END_RUNG wire#w1
   // the same network as SCL:
   #SWITCH_OFF_GLOBAL_REQUEST := (#SWITCH_OFF_MANUAL_REQUEST AND "DB2001_MODES_GENERAL".GENERAL.MANUAL_SELECTED) OR (#SWITCH_OFF_AUTO_REQUEST AND "DB2001_MODES_GENERAL".GENERAL.AUTO_SINGLE_SEMI_SELECTED) OR NOT (NOT "DB2120_MPP_ITC_IPC".STOP_SERVICES_GLOBAL);
END_REGION

REGION Network 22: SWITCH OFF COMMAND
   RUNG wire#powerrail
      Contact( #SWITCH_OFF_GLOBAL_REQUEST )
      Contact( #SWITCH_OFF_GENERAL_CONDITIONS )
      Contact( #SWITCH_OFF_INITIAL_CONDITIONS )
      Coil( #SWITCH_OFF_COMMAND )
   END_RUNG
   // the same network as SCL:
   #SWITCH_OFF_COMMAND := #SWITCH_OFF_GLOBAL_REQUEST AND #SWITCH_OFF_GENERAL_CONDITIONS AND #SWITCH_OFF_INITIAL_CONDITIONS;
END_REGION

REGION Network 23: OUT OF SERVICE
   RUNG wire#powerrail
      I_Contact( #IN_SERVICE )
      Coil( #OUT_OF_SERVICE )
   END_RUNG
   // the same network as SCL:
   #OUT_OF_SERVICE := NOT #IN_SERVICE;
END_REGION

REGION Network 24: UNIT 01 & UNIT 02 CIRCUIT BREAKER TRIPPED ALARM
   RUNG wire#powerrail
      Contact( #CIRCUIT_BREAKER_INPUT )
      wire#w1
      Contact( "DB2120_MPP_ITC_IPC".MACHINE_ON_DELAYED )
      Contact( #O_BYTE_0.GEN_CIRCUIT_BREAKER )
      Coil( #U01_U02_BREAKER_TRIPPED_ALARM )
   END_RUNG
   RUNG wire#powerrail
      Contact( #U01_U02_BREAKER_TRIPPED_ALARM )
      I_Contact( "DB2120_MPP_ITC_IPC".RESET_FAULTS )
   END_RUNG wire#w1
   // the same network as SCL:
   #U01_U02_BREAKER_TRIPPED_ALARM := (#CIRCUIT_BREAKER_INPUT OR (#U01_U02_BREAKER_TRIPPED_ALARM AND NOT "DB2120_MPP_ITC_IPC".RESET_FAULTS)) AND "DB2120_MPP_ITC_IPC".MACHINE_ON_DELAYED AND #O_BYTE_0.GEN_CIRCUIT_BREAKER;
END_REGION

REGION Network 25: UNIT 01 & UNIT 02 CONTACTOR FEEDBACK ALARM / MAIN CHIP CONVEYOR FORWARD FEEDBACK
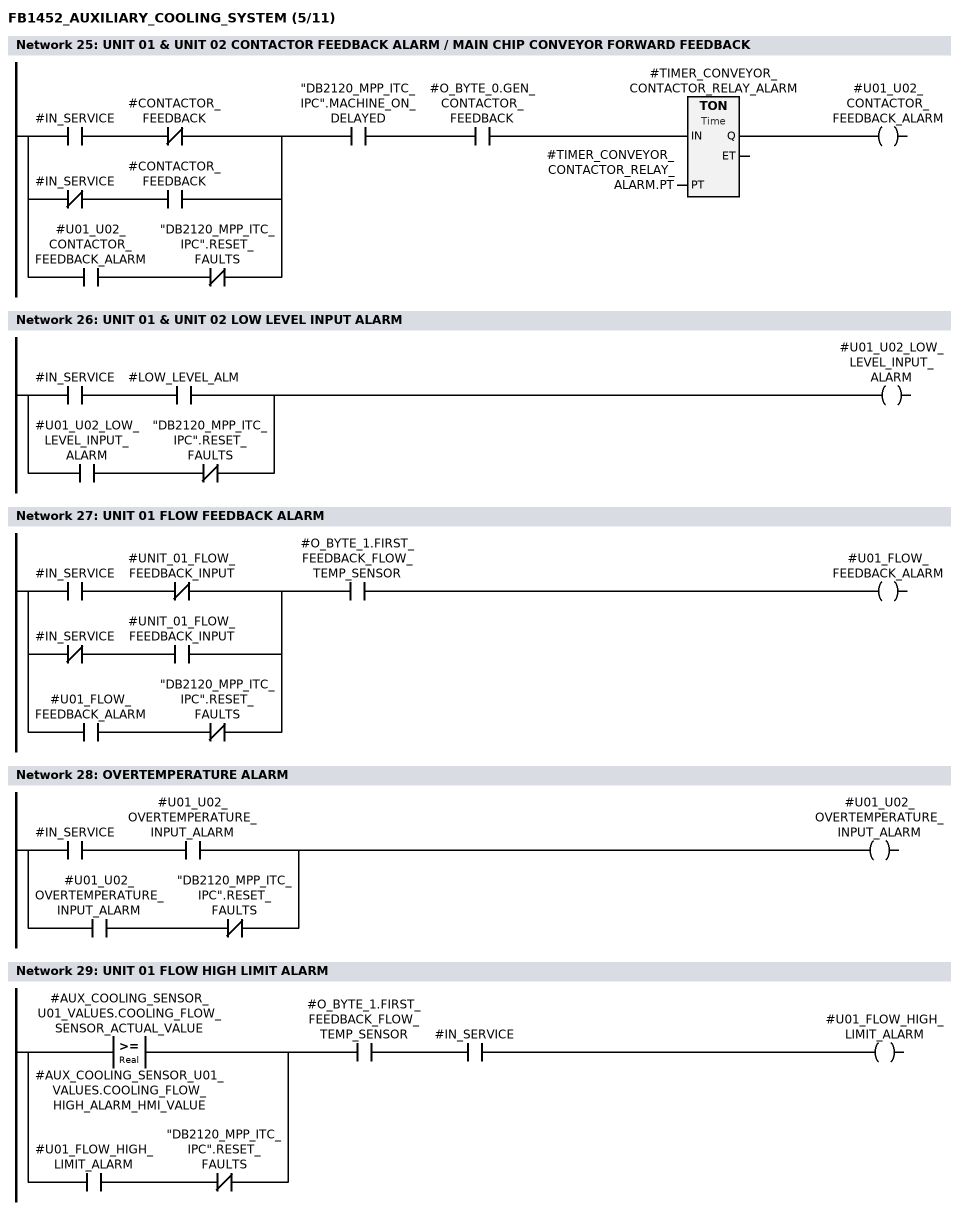
   RUNG wire#powerrail
      Contact( #IN_SERVICE )
      I_Contact( #CONTACTOR_FEEDBACK )
      wire#w1
      Contact( "DB2120_MPP_ITC_IPC".MACHINE_ON_DELAYED )
      Contact( #O_BYTE_0.GEN_CONTACTOR_FEEDBACK )
      { S7_Templates := "time_type := Time" } #TIMER_CONVEYOR_CONTACTOR_RELAY_ALARM.TON(pt := #TIMER_CONVEYOR_CONTACTOR_RELAY_ALARM.PT, et =>)
      Coil( #U01_U02_CONTACTOR_FEEDBACK_ALARM )
   END_RUNG
   RUNG wire#powerrail
      I_Contact( #IN_SERVICE )
      Contact( #CONTACTOR_FEEDBACK )
   END_RUNG wire#w1
   RUNG wire#powerrail
      Contact( #U01_U02_CONTACTOR_FEEDBACK_ALARM )
      I_Contact( "DB2120_MPP_ITC_IPC".RESET_FAULTS )
   END_RUNG wire#w1
   // the same network as SCL:
   #TIMER_CONVEYOR_CONTACTOR_RELAY_ALARM(IN := ((#IN_SERVICE AND NOT #CONTACTOR_FEEDBACK) OR (NOT #IN_SERVICE AND #CONTACTOR_FEEDBACK) OR (#U01_U02_CONTACTOR_FEEDBACK_ALARM AND NOT "DB2120_MPP_ITC_IPC".RESET_FAULTS)) AND "DB2120_MPP_ITC_IPC".MACHINE_ON_DELAYED AND #O_BYTE_0.GEN_CONTACTOR_FEEDBACK,   // TON
                           PT := #TIMER_CONVEYOR_CONTACTOR_RELAY_ALARM.PT);
   #U01_U02_CONTACTOR_FEEDBACK_ALARM := #TIMER_CONVEYOR_CONTACTOR_RELAY_ALARM.Q;
END_REGION

REGION Network 26: UNIT 01 & UNIT 02 LOW LEVEL INPUT ALARM
   RUNG wire#powerrail
      Contact( #IN_SERVICE )
      Contact( #LOW_LEVEL_ALM )
      wire#w1
      Coil( #U01_U02_LOW_LEVEL_INPUT_ALARM )
   END_RUNG
   RUNG wire#powerrail
      Contact( #U01_U02_LOW_LEVEL_INPUT_ALARM )
      I_Contact( "DB2120_MPP_ITC_IPC".RESET_FAULTS )
   END_RUNG wire#w1
   // the same network as SCL:
   #U01_U02_LOW_LEVEL_INPUT_ALARM := (#IN_SERVICE AND #LOW_LEVEL_ALM) OR (#U01_U02_LOW_LEVEL_INPUT_ALARM AND NOT "DB2120_MPP_ITC_IPC".RESET_FAULTS);
END_REGION

REGION Network 27: UNIT 01 FLOW FEEDBACK ALARM
   RUNG wire#powerrail
      Contact( #IN_SERVICE )
      I_Contact( #UNIT_01_FLOW_FEEDBACK_INPUT )
      wire#w1
      Contact( #O_BYTE_1.FIRST_FEEDBACK_FLOW_TEMP_SENSOR )
      Coil( #U01_FLOW_FEEDBACK_ALARM )
   END_RUNG
   RUNG wire#powerrail
      I_Contact( #IN_SERVICE )
      Contact( #UNIT_01_FLOW_FEEDBACK_INPUT )
   END_RUNG wire#w1
   RUNG wire#powerrail
      Contact( #U01_FLOW_FEEDBACK_ALARM )
      I_Contact( "DB2120_MPP_ITC_IPC".RESET_FAULTS )
   END_RUNG wire#w1
   // the same network as SCL:
   #U01_FLOW_FEEDBACK_ALARM := ((#IN_SERVICE AND NOT #UNIT_01_FLOW_FEEDBACK_INPUT) OR (NOT #IN_SERVICE AND #UNIT_01_FLOW_FEEDBACK_INPUT) OR (#U01_FLOW_FEEDBACK_ALARM AND NOT "DB2120_MPP_ITC_IPC".RESET_FAULTS)) AND #O_BYTE_1.FIRST_FEEDBACK_FLOW_TEMP_SENSOR;
END_REGION

REGION Network 28: OVERTEMPERATURE ALARM
   RUNG wire#powerrail
      Contact( #IN_SERVICE )
      Contact( #U01_U02_OVERTEMPERATURE_INPUT_ALARM )
      wire#w1
      Coil( #U01_U02_OVERTEMPERATURE_INPUT_ALARM )
   END_RUNG
   RUNG wire#powerrail
      Contact( #U01_U02_OVERTEMPERATURE_INPUT_ALARM )
      I_Contact( "DB2120_MPP_ITC_IPC".RESET_FAULTS )
   END_RUNG wire#w1
   // the same network as SCL:
   #U01_U02_OVERTEMPERATURE_INPUT_ALARM := (#IN_SERVICE AND #U01_U02_OVERTEMPERATURE_INPUT_ALARM) OR (#U01_U02_OVERTEMPERATURE_INPUT_ALARM AND NOT "DB2120_MPP_ITC_IPC".RESET_FAULTS);
END_REGION

REGION Network 29: UNIT 01 FLOW HIGH LIMIT ALARM
   RUNG wire#powerrail
      { S7_Templates := "SrcType := Real" } GE_Contact(in1 := #AUX_COOLING_SENSOR_U01_VALUES.COOLING_FLOW_SENSOR_ACTUAL_VALUE, in2 := #AUX_COOLING_SENSOR_U01_VALUES.COOLING_FLOW_HIGH_ALARM_HMI_VALUE)
      wire#w1
      Contact( #O_BYTE_1.FIRST_FEEDBACK_FLOW_TEMP_SENSOR )
      Contact( #IN_SERVICE )
      Coil( #U01_FLOW_HIGH_LIMIT_ALARM )
   END_RUNG
   RUNG wire#powerrail
      Contact( #U01_FLOW_HIGH_LIMIT_ALARM )
      I_Contact( "DB2120_MPP_ITC_IPC".RESET_FAULTS )
   END_RUNG wire#w1
   // the same network as SCL:
   #U01_FLOW_HIGH_LIMIT_ALARM := ((#AUX_COOLING_SENSOR_U01_VALUES.COOLING_FLOW_SENSOR_ACTUAL_VALUE >= #AUX_COOLING_SENSOR_U01_VALUES.COOLING_FLOW_HIGH_ALARM_HMI_VALUE) OR (#U01_FLOW_HIGH_LIMIT_ALARM AND NOT "DB2120_MPP_ITC_IPC".RESET_FAULTS)) AND #O_BYTE_1.FIRST_FEEDBACK_FLOW_TEMP_SENSOR AND #IN_SERVICE;
END_REGION

REGION Network 30: UNIT 01 FLOW HIGH LIMIT WARNING
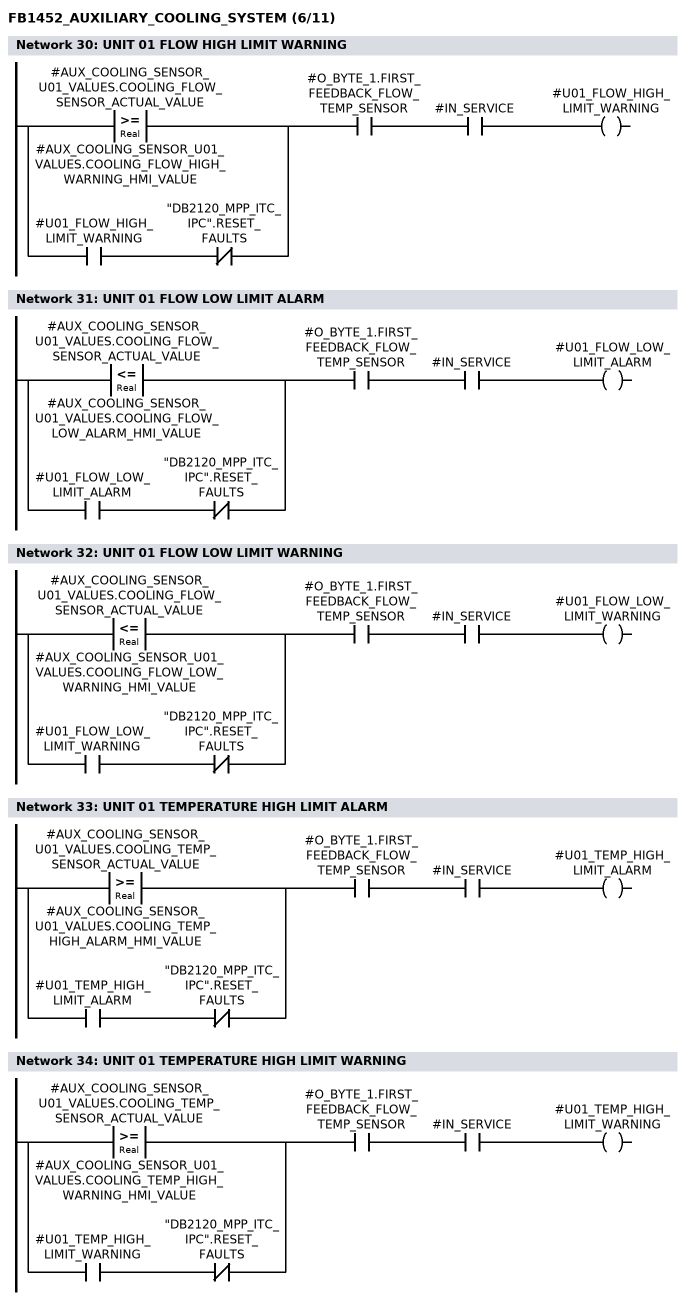
   RUNG wire#powerrail
      { S7_Templates := "SrcType := Real" } GE_Contact(in1 := #AUX_COOLING_SENSOR_U01_VALUES.COOLING_FLOW_SENSOR_ACTUAL_VALUE, in2 := #AUX_COOLING_SENSOR_U01_VALUES.COOLING_FLOW_HIGH_WARNING_HMI_VALUE)
      wire#w1
      Contact( #O_BYTE_1.FIRST_FEEDBACK_FLOW_TEMP_SENSOR )
      Contact( #IN_SERVICE )
      Coil( #U01_FLOW_HIGH_LIMIT_WARNING )
   END_RUNG
   RUNG wire#powerrail
      Contact( #U01_FLOW_HIGH_LIMIT_WARNING )
      I_Contact( "DB2120_MPP_ITC_IPC".RESET_FAULTS )
   END_RUNG wire#w1
   // the same network as SCL:
   #U01_FLOW_HIGH_LIMIT_WARNING := ((#AUX_COOLING_SENSOR_U01_VALUES.COOLING_FLOW_SENSOR_ACTUAL_VALUE >= #AUX_COOLING_SENSOR_U01_VALUES.COOLING_FLOW_HIGH_WARNING_HMI_VALUE) OR (#U01_FLOW_HIGH_LIMIT_WARNING AND NOT "DB2120_MPP_ITC_IPC".RESET_FAULTS)) AND #O_BYTE_1.FIRST_FEEDBACK_FLOW_TEMP_SENSOR AND #IN_SERVICE;
END_REGION

REGION Network 31: UNIT 01 FLOW LOW LIMIT ALARM
   RUNG wire#powerrail
      { S7_Templates := "SrcType := Real" } LE_Contact(in1 := #AUX_COOLING_SENSOR_U01_VALUES.COOLING_FLOW_SENSOR_ACTUAL_VALUE, in2 := #AUX_COOLING_SENSOR_U01_VALUES.COOLING_FLOW_LOW_ALARM_HMI_VALUE)
      wire#w1
      Contact( #O_BYTE_1.FIRST_FEEDBACK_FLOW_TEMP_SENSOR )
      Contact( #IN_SERVICE )
      Coil( #U01_FLOW_LOW_LIMIT_ALARM )
   END_RUNG
   RUNG wire#powerrail
      Contact( #U01_FLOW_LOW_LIMIT_ALARM )
      I_Contact( "DB2120_MPP_ITC_IPC".RESET_FAULTS )
   END_RUNG wire#w1
   // the same network as SCL:
   #U01_FLOW_LOW_LIMIT_ALARM := ((#AUX_COOLING_SENSOR_U01_VALUES.COOLING_FLOW_SENSOR_ACTUAL_VALUE <= #AUX_COOLING_SENSOR_U01_VALUES.COOLING_FLOW_LOW_ALARM_HMI_VALUE) OR (#U01_FLOW_LOW_LIMIT_ALARM AND NOT "DB2120_MPP_ITC_IPC".RESET_FAULTS)) AND #O_BYTE_1.FIRST_FEEDBACK_FLOW_TEMP_SENSOR AND #IN_SERVICE;
END_REGION

REGION Network 32: UNIT 01 FLOW LOW LIMIT WARNING
   RUNG wire#powerrail
      { S7_Templates := "SrcType := Real" } LE_Contact(in1 := #AUX_COOLING_SENSOR_U01_VALUES.COOLING_FLOW_SENSOR_ACTUAL_VALUE, in2 := #AUX_COOLING_SENSOR_U01_VALUES.COOLING_FLOW_LOW_WARNING_HMI_VALUE)
      wire#w1
      Contact( #O_BYTE_1.FIRST_FEEDBACK_FLOW_TEMP_SENSOR )
      Contact( #IN_SERVICE )
      Coil( #U01_FLOW_LOW_LIMIT_WARNING )
   END_RUNG
   RUNG wire#powerrail
      Contact( #U01_FLOW_LOW_LIMIT_WARNING )
      I_Contact( "DB2120_MPP_ITC_IPC".RESET_FAULTS )
   END_RUNG wire#w1
   // the same network as SCL:
   #U01_FLOW_LOW_LIMIT_WARNING := ((#AUX_COOLING_SENSOR_U01_VALUES.COOLING_FLOW_SENSOR_ACTUAL_VALUE <= #AUX_COOLING_SENSOR_U01_VALUES.COOLING_FLOW_LOW_WARNING_HMI_VALUE) OR (#U01_FLOW_LOW_LIMIT_WARNING AND NOT "DB2120_MPP_ITC_IPC".RESET_FAULTS)) AND #O_BYTE_1.FIRST_FEEDBACK_FLOW_TEMP_SENSOR AND #IN_SERVICE;
END_REGION

REGION Network 33: UNIT 01 TEMPERATURE HIGH LIMIT ALARM
   RUNG wire#powerrail
      { S7_Templates := "SrcType := Real" } GE_Contact(in1 := #AUX_COOLING_SENSOR_U01_VALUES.COOLING_TEMP_SENSOR_ACTUAL_VALUE, in2 := #AUX_COOLING_SENSOR_U01_VALUES.COOLING_TEMP_HIGH_ALARM_HMI_VALUE)
      wire#w1
      Contact( #O_BYTE_1.FIRST_FEEDBACK_FLOW_TEMP_SENSOR )
      Contact( #IN_SERVICE )
      Coil( #U01_TEMP_HIGH_LIMIT_ALARM )
   END_RUNG
   RUNG wire#powerrail
      Contact( #U01_TEMP_HIGH_LIMIT_ALARM )
      I_Contact( "DB2120_MPP_ITC_IPC".RESET_FAULTS )
   END_RUNG wire#w1
   // the same network as SCL:
   #U01_TEMP_HIGH_LIMIT_ALARM := ((#AUX_COOLING_SENSOR_U01_VALUES.COOLING_TEMP_SENSOR_ACTUAL_VALUE >= #AUX_COOLING_SENSOR_U01_VALUES.COOLING_TEMP_HIGH_ALARM_HMI_VALUE) OR (#U01_TEMP_HIGH_LIMIT_ALARM AND NOT "DB2120_MPP_ITC_IPC".RESET_FAULTS)) AND #O_BYTE_1.FIRST_FEEDBACK_FLOW_TEMP_SENSOR AND #IN_SERVICE;
END_REGION

REGION Network 34: UNIT 01 TEMPERATURE HIGH LIMIT WARNING
   RUNG wire#powerrail
      { S7_Templates := "SrcType := Real" } GE_Contact(in1 := #AUX_COOLING_SENSOR_U01_VALUES.COOLING_TEMP_SENSOR_ACTUAL_VALUE, in2 := #AUX_COOLING_SENSOR_U01_VALUES.COOLING_TEMP_HIGH_WARNING_HMI_VALUE)
      wire#w1
      Contact( #O_BYTE_1.FIRST_FEEDBACK_FLOW_TEMP_SENSOR )
      Contact( #IN_SERVICE )
      Coil( #U01_TEMP_HIGH_LIMIT_WARNING )
   END_RUNG
   RUNG wire#powerrail
      Contact( #U01_TEMP_HIGH_LIMIT_WARNING )
      I_Contact( "DB2120_MPP_ITC_IPC".RESET_FAULTS )
   END_RUNG wire#w1
   // the same network as SCL:
   #U01_TEMP_HIGH_LIMIT_WARNING := ((#AUX_COOLING_SENSOR_U01_VALUES.COOLING_TEMP_SENSOR_ACTUAL_VALUE >= #AUX_COOLING_SENSOR_U01_VALUES.COOLING_TEMP_HIGH_WARNING_HMI_VALUE) OR (#U01_TEMP_HIGH_LIMIT_WARNING AND NOT "DB2120_MPP_ITC_IPC".RESET_FAULTS)) AND #O_BYTE_1.FIRST_FEEDBACK_FLOW_TEMP_SENSOR AND #IN_SERVICE;
END_REGION

REGION Network 35: UNIT 01 TEMPERATURE LOW LIMIT ALARM
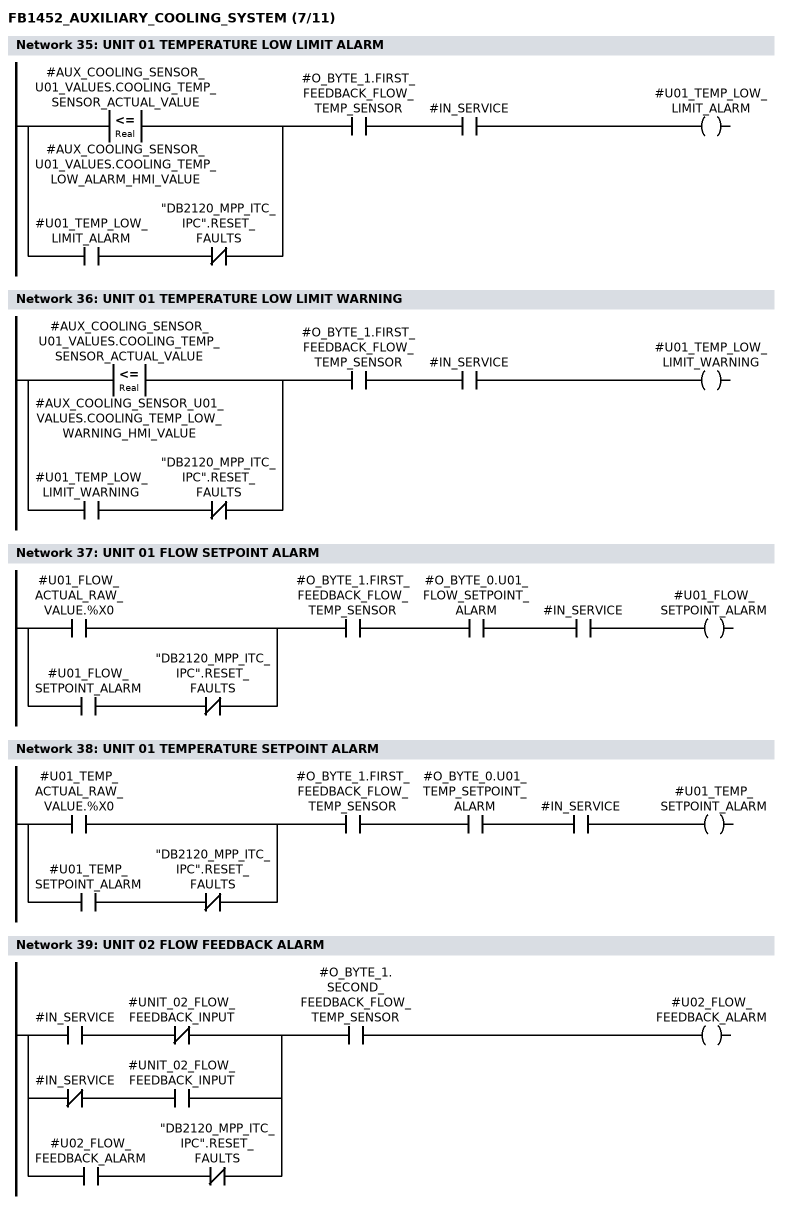
   RUNG wire#powerrail
      { S7_Templates := "SrcType := Real" } LE_Contact(in1 := #AUX_COOLING_SENSOR_U01_VALUES.COOLING_TEMP_SENSOR_ACTUAL_VALUE, in2 := #AUX_COOLING_SENSOR_U01_VALUES.COOLING_TEMP_LOW_ALARM_HMI_VALUE)
      wire#w1
      Contact( #O_BYTE_1.FIRST_FEEDBACK_FLOW_TEMP_SENSOR )
      Contact( #IN_SERVICE )
      Coil( #U01_TEMP_LOW_LIMIT_ALARM )
   END_RUNG
   RUNG wire#powerrail
      Contact( #U01_TEMP_LOW_LIMIT_ALARM )
      I_Contact( "DB2120_MPP_ITC_IPC".RESET_FAULTS )
   END_RUNG wire#w1
   // the same network as SCL:
   #U01_TEMP_LOW_LIMIT_ALARM := ((#AUX_COOLING_SENSOR_U01_VALUES.COOLING_TEMP_SENSOR_ACTUAL_VALUE <= #AUX_COOLING_SENSOR_U01_VALUES.COOLING_TEMP_LOW_ALARM_HMI_VALUE) OR (#U01_TEMP_LOW_LIMIT_ALARM AND NOT "DB2120_MPP_ITC_IPC".RESET_FAULTS)) AND #O_BYTE_1.FIRST_FEEDBACK_FLOW_TEMP_SENSOR AND #IN_SERVICE;
END_REGION

REGION Network 36: UNIT 01 TEMPERATURE LOW LIMIT WARNING
   RUNG wire#powerrail
      { S7_Templates := "SrcType := Real" } LE_Contact(in1 := #AUX_COOLING_SENSOR_U01_VALUES.COOLING_TEMP_SENSOR_ACTUAL_VALUE, in2 := #AUX_COOLING_SENSOR_U01_VALUES.COOLING_TEMP_LOW_WARNING_HMI_VALUE)
      wire#w1
      Contact( #O_BYTE_1.FIRST_FEEDBACK_FLOW_TEMP_SENSOR )
      Contact( #IN_SERVICE )
      Coil( #U01_TEMP_LOW_LIMIT_WARNING )
   END_RUNG
   RUNG wire#powerrail
      Contact( #U01_TEMP_LOW_LIMIT_WARNING )
      I_Contact( "DB2120_MPP_ITC_IPC".RESET_FAULTS )
   END_RUNG wire#w1
   // the same network as SCL:
   #U01_TEMP_LOW_LIMIT_WARNING := ((#AUX_COOLING_SENSOR_U01_VALUES.COOLING_TEMP_SENSOR_ACTUAL_VALUE <= #AUX_COOLING_SENSOR_U01_VALUES.COOLING_TEMP_LOW_WARNING_HMI_VALUE) OR (#U01_TEMP_LOW_LIMIT_WARNING AND NOT "DB2120_MPP_ITC_IPC".RESET_FAULTS)) AND #O_BYTE_1.FIRST_FEEDBACK_FLOW_TEMP_SENSOR AND #IN_SERVICE;
END_REGION

REGION Network 37: UNIT 01 FLOW SETPOINT ALARM
   RUNG wire#powerrail
      Contact( #U01_FLOW_ACTUAL_RAW_VALUE.%X0 )
      wire#w1
      Contact( #O_BYTE_1.FIRST_FEEDBACK_FLOW_TEMP_SENSOR )
      Contact( #O_BYTE_0.U01_FLOW_SETPOINT_ALARM )
      Contact( #IN_SERVICE )
      Coil( #U01_FLOW_SETPOINT_ALARM )
   END_RUNG
   RUNG wire#powerrail
      Contact( #U01_FLOW_SETPOINT_ALARM )
      I_Contact( "DB2120_MPP_ITC_IPC".RESET_FAULTS )
   END_RUNG wire#w1
   // the same network as SCL:
   #U01_FLOW_SETPOINT_ALARM := (#U01_FLOW_ACTUAL_RAW_VALUE.%X0 OR (#U01_FLOW_SETPOINT_ALARM AND NOT "DB2120_MPP_ITC_IPC".RESET_FAULTS)) AND #O_BYTE_1.FIRST_FEEDBACK_FLOW_TEMP_SENSOR AND #O_BYTE_0.U01_FLOW_SETPOINT_ALARM AND #IN_SERVICE;
END_REGION

REGION Network 38: UNIT 01 TEMPERATURE SETPOINT ALARM
   RUNG wire#powerrail
      Contact( #U01_TEMP_ACTUAL_RAW_VALUE.%X0 )
      wire#w1
      Contact( #O_BYTE_1.FIRST_FEEDBACK_FLOW_TEMP_SENSOR )
      Contact( #O_BYTE_0.U01_TEMP_SETPOINT_ALARM )
      Contact( #IN_SERVICE )
      Coil( #U01_TEMP_SETPOINT_ALARM )
   END_RUNG
   RUNG wire#powerrail
      Contact( #U01_TEMP_SETPOINT_ALARM )
      I_Contact( "DB2120_MPP_ITC_IPC".RESET_FAULTS )
   END_RUNG wire#w1
   // the same network as SCL:
   #U01_TEMP_SETPOINT_ALARM := (#U01_TEMP_ACTUAL_RAW_VALUE.%X0 OR (#U01_TEMP_SETPOINT_ALARM AND NOT "DB2120_MPP_ITC_IPC".RESET_FAULTS)) AND #O_BYTE_1.FIRST_FEEDBACK_FLOW_TEMP_SENSOR AND #O_BYTE_0.U01_TEMP_SETPOINT_ALARM AND #IN_SERVICE;
END_REGION

REGION Network 39: UNIT 02 FLOW FEEDBACK ALARM
   RUNG wire#powerrail
      Contact( #IN_SERVICE )
      I_Contact( #UNIT_02_FLOW_FEEDBACK_INPUT )
      wire#w1
      Contact( #O_BYTE_1.SECOND_FEEDBACK_FLOW_TEMP_SENSOR )
      Coil( #U02_FLOW_FEEDBACK_ALARM )
   END_RUNG
   RUNG wire#powerrail
      I_Contact( #IN_SERVICE )
      Contact( #UNIT_02_FLOW_FEEDBACK_INPUT )
   END_RUNG wire#w1
   RUNG wire#powerrail
      Contact( #U02_FLOW_FEEDBACK_ALARM )
      I_Contact( "DB2120_MPP_ITC_IPC".RESET_FAULTS )
   END_RUNG wire#w1
   // the same network as SCL:
   #U02_FLOW_FEEDBACK_ALARM := ((#IN_SERVICE AND NOT #UNIT_02_FLOW_FEEDBACK_INPUT) OR (NOT #IN_SERVICE AND #UNIT_02_FLOW_FEEDBACK_INPUT) OR (#U02_FLOW_FEEDBACK_ALARM AND NOT "DB2120_MPP_ITC_IPC".RESET_FAULTS)) AND #O_BYTE_1.SECOND_FEEDBACK_FLOW_TEMP_SENSOR;
END_REGION

REGION Network 40: UNIT 02 FLOW HIGH LIMIT ALARM
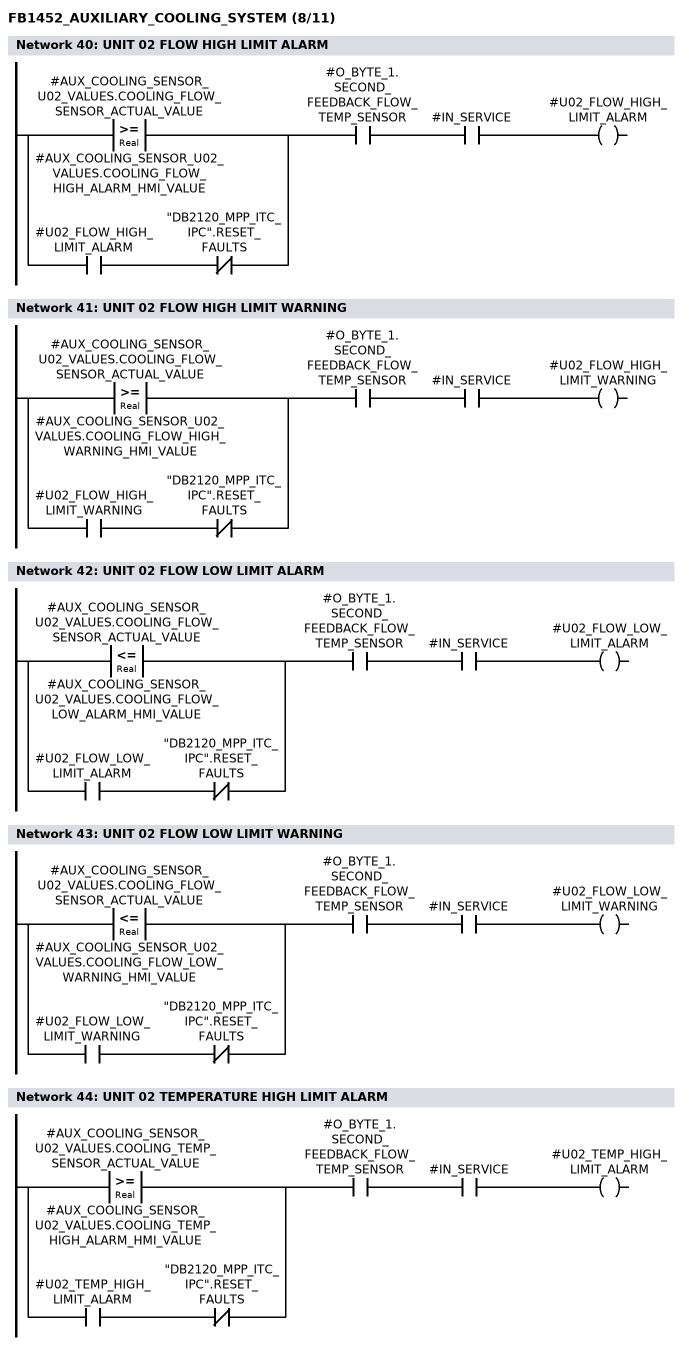
   RUNG wire#powerrail
      { S7_Templates := "SrcType := Real" } GE_Contact(in1 := #AUX_COOLING_SENSOR_U02_VALUES.COOLING_FLOW_SENSOR_ACTUAL_VALUE, in2 := #AUX_COOLING_SENSOR_U02_VALUES.COOLING_FLOW_HIGH_ALARM_HMI_VALUE)
      wire#w1
      Contact( #O_BYTE_1.SECOND_FEEDBACK_FLOW_TEMP_SENSOR )
      Contact( #IN_SERVICE )
      Coil( #U02_FLOW_HIGH_LIMIT_ALARM )
   END_RUNG
   RUNG wire#powerrail
      Contact( #U02_FLOW_HIGH_LIMIT_ALARM )
      I_Contact( "DB2120_MPP_ITC_IPC".RESET_FAULTS )
   END_RUNG wire#w1
   // the same network as SCL:
   #U02_FLOW_HIGH_LIMIT_ALARM := ((#AUX_COOLING_SENSOR_U02_VALUES.COOLING_FLOW_SENSOR_ACTUAL_VALUE >= #AUX_COOLING_SENSOR_U02_VALUES.COOLING_FLOW_HIGH_ALARM_HMI_VALUE) OR (#U02_FLOW_HIGH_LIMIT_ALARM AND NOT "DB2120_MPP_ITC_IPC".RESET_FAULTS)) AND #O_BYTE_1.SECOND_FEEDBACK_FLOW_TEMP_SENSOR AND #IN_SERVICE;
END_REGION

REGION Network 41: UNIT 02 FLOW HIGH LIMIT WARNING
   RUNG wire#powerrail
      { S7_Templates := "SrcType := Real" } GE_Contact(in1 := #AUX_COOLING_SENSOR_U02_VALUES.COOLING_FLOW_SENSOR_ACTUAL_VALUE, in2 := #AUX_COOLING_SENSOR_U02_VALUES.COOLING_FLOW_HIGH_WARNING_HMI_VALUE)
      wire#w1
      Contact( #O_BYTE_1.SECOND_FEEDBACK_FLOW_TEMP_SENSOR )
      Contact( #IN_SERVICE )
      Coil( #U02_FLOW_HIGH_LIMIT_WARNING )
   END_RUNG
   RUNG wire#powerrail
      Contact( #U02_FLOW_HIGH_LIMIT_WARNING )
      I_Contact( "DB2120_MPP_ITC_IPC".RESET_FAULTS )
   END_RUNG wire#w1
   // the same network as SCL:
   #U02_FLOW_HIGH_LIMIT_WARNING := ((#AUX_COOLING_SENSOR_U02_VALUES.COOLING_FLOW_SENSOR_ACTUAL_VALUE >= #AUX_COOLING_SENSOR_U02_VALUES.COOLING_FLOW_HIGH_WARNING_HMI_VALUE) OR (#U02_FLOW_HIGH_LIMIT_WARNING AND NOT "DB2120_MPP_ITC_IPC".RESET_FAULTS)) AND #O_BYTE_1.SECOND_FEEDBACK_FLOW_TEMP_SENSOR AND #IN_SERVICE;
END_REGION

REGION Network 42: UNIT 02 FLOW LOW LIMIT ALARM
   RUNG wire#powerrail
      { S7_Templates := "SrcType := Real" } LE_Contact(in1 := #AUX_COOLING_SENSOR_U02_VALUES.COOLING_FLOW_SENSOR_ACTUAL_VALUE, in2 := #AUX_COOLING_SENSOR_U02_VALUES.COOLING_FLOW_LOW_ALARM_HMI_VALUE)
      wire#w1
      Contact( #O_BYTE_1.SECOND_FEEDBACK_FLOW_TEMP_SENSOR )
      Contact( #IN_SERVICE )
      Coil( #U02_FLOW_LOW_LIMIT_ALARM )
   END_RUNG
   RUNG wire#powerrail
      Contact( #U02_FLOW_LOW_LIMIT_ALARM )
      I_Contact( "DB2120_MPP_ITC_IPC".RESET_FAULTS )
   END_RUNG wire#w1
   // the same network as SCL:
   #U02_FLOW_LOW_LIMIT_ALARM := ((#AUX_COOLING_SENSOR_U02_VALUES.COOLING_FLOW_SENSOR_ACTUAL_VALUE <= #AUX_COOLING_SENSOR_U02_VALUES.COOLING_FLOW_LOW_ALARM_HMI_VALUE) OR (#U02_FLOW_LOW_LIMIT_ALARM AND NOT "DB2120_MPP_ITC_IPC".RESET_FAULTS)) AND #O_BYTE_1.SECOND_FEEDBACK_FLOW_TEMP_SENSOR AND #IN_SERVICE;
END_REGION

REGION Network 43: UNIT 02 FLOW LOW LIMIT WARNING
   RUNG wire#powerrail
      { S7_Templates := "SrcType := Real" } LE_Contact(in1 := #AUX_COOLING_SENSOR_U02_VALUES.COOLING_FLOW_SENSOR_ACTUAL_VALUE, in2 := #AUX_COOLING_SENSOR_U02_VALUES.COOLING_FLOW_LOW_WARNING_HMI_VALUE)
      wire#w1
      Contact( #O_BYTE_1.SECOND_FEEDBACK_FLOW_TEMP_SENSOR )
      Contact( #IN_SERVICE )
      Coil( #U02_FLOW_LOW_LIMIT_WARNING )
   END_RUNG
   RUNG wire#powerrail
      Contact( #U02_FLOW_LOW_LIMIT_WARNING )
      I_Contact( "DB2120_MPP_ITC_IPC".RESET_FAULTS )
   END_RUNG wire#w1
   // the same network as SCL:
   #U02_FLOW_LOW_LIMIT_WARNING := ((#AUX_COOLING_SENSOR_U02_VALUES.COOLING_FLOW_SENSOR_ACTUAL_VALUE <= #AUX_COOLING_SENSOR_U02_VALUES.COOLING_FLOW_LOW_WARNING_HMI_VALUE) OR (#U02_FLOW_LOW_LIMIT_WARNING AND NOT "DB2120_MPP_ITC_IPC".RESET_FAULTS)) AND #O_BYTE_1.SECOND_FEEDBACK_FLOW_TEMP_SENSOR AND #IN_SERVICE;
END_REGION

REGION Network 44: UNIT 02 TEMPERATURE HIGH LIMIT ALARM
   RUNG wire#powerrail
      { S7_Templates := "SrcType := Real" } GE_Contact(in1 := #AUX_COOLING_SENSOR_U02_VALUES.COOLING_TEMP_SENSOR_ACTUAL_VALUE, in2 := #AUX_COOLING_SENSOR_U02_VALUES.COOLING_TEMP_HIGH_ALARM_HMI_VALUE)
      wire#w1
      Contact( #O_BYTE_1.SECOND_FEEDBACK_FLOW_TEMP_SENSOR )
      Contact( #IN_SERVICE )
      Coil( #U02_TEMP_HIGH_LIMIT_ALARM )
   END_RUNG
   RUNG wire#powerrail
      Contact( #U02_TEMP_HIGH_LIMIT_ALARM )
      I_Contact( "DB2120_MPP_ITC_IPC".RESET_FAULTS )
   END_RUNG wire#w1
   // the same network as SCL:
   #U02_TEMP_HIGH_LIMIT_ALARM := ((#AUX_COOLING_SENSOR_U02_VALUES.COOLING_TEMP_SENSOR_ACTUAL_VALUE >= #AUX_COOLING_SENSOR_U02_VALUES.COOLING_TEMP_HIGH_ALARM_HMI_VALUE) OR (#U02_TEMP_HIGH_LIMIT_ALARM AND NOT "DB2120_MPP_ITC_IPC".RESET_FAULTS)) AND #O_BYTE_1.SECOND_FEEDBACK_FLOW_TEMP_SENSOR AND #IN_SERVICE;
END_REGION

REGION Network 45: UNIT 02 TEMPERATURE HIGH LIMIT WARNING
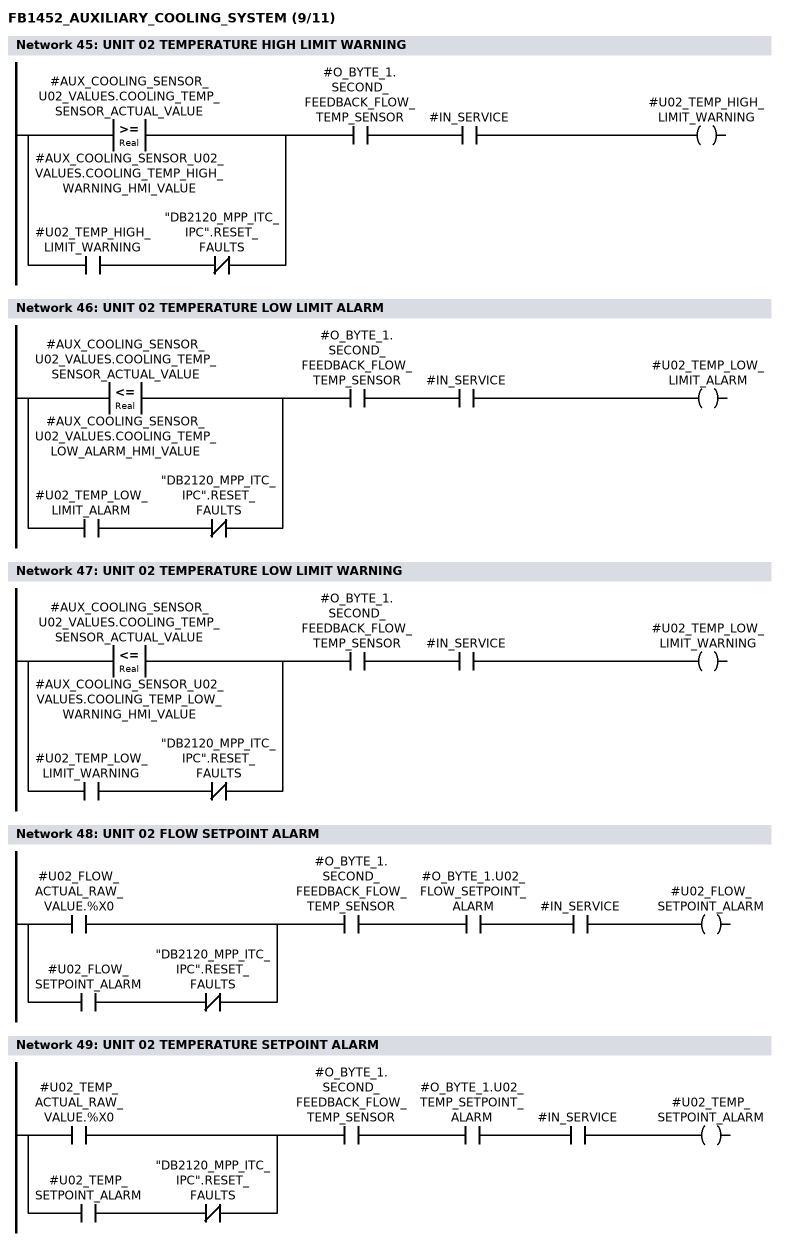
   RUNG wire#powerrail
      { S7_Templates := "SrcType := Real" } GE_Contact(in1 := #AUX_COOLING_SENSOR_U02_VALUES.COOLING_TEMP_SENSOR_ACTUAL_VALUE, in2 := #AUX_COOLING_SENSOR_U02_VALUES.COOLING_TEMP_HIGH_WARNING_HMI_VALUE)
      wire#w1
      Contact( #O_BYTE_1.SECOND_FEEDBACK_FLOW_TEMP_SENSOR )
      Contact( #IN_SERVICE )
      Coil( #U02_TEMP_HIGH_LIMIT_WARNING )
   END_RUNG
   RUNG wire#powerrail
      Contact( #U02_TEMP_HIGH_LIMIT_WARNING )
      I_Contact( "DB2120_MPP_ITC_IPC".RESET_FAULTS )
   END_RUNG wire#w1
   // the same network as SCL:
   #U02_TEMP_HIGH_LIMIT_WARNING := ((#AUX_COOLING_SENSOR_U02_VALUES.COOLING_TEMP_SENSOR_ACTUAL_VALUE >= #AUX_COOLING_SENSOR_U02_VALUES.COOLING_TEMP_HIGH_WARNING_HMI_VALUE) OR (#U02_TEMP_HIGH_LIMIT_WARNING AND NOT "DB2120_MPP_ITC_IPC".RESET_FAULTS)) AND #O_BYTE_1.SECOND_FEEDBACK_FLOW_TEMP_SENSOR AND #IN_SERVICE;
END_REGION

REGION Network 46: UNIT 02 TEMPERATURE LOW LIMIT ALARM
   RUNG wire#powerrail
      { S7_Templates := "SrcType := Real" } LE_Contact(in1 := #AUX_COOLING_SENSOR_U02_VALUES.COOLING_TEMP_SENSOR_ACTUAL_VALUE, in2 := #AUX_COOLING_SENSOR_U02_VALUES.COOLING_TEMP_LOW_ALARM_HMI_VALUE)
      wire#w1
      Contact( #O_BYTE_1.SECOND_FEEDBACK_FLOW_TEMP_SENSOR )
      Contact( #IN_SERVICE )
      Coil( #U02_TEMP_LOW_LIMIT_ALARM )
   END_RUNG
   RUNG wire#powerrail
      Contact( #U02_TEMP_LOW_LIMIT_ALARM )
      I_Contact( "DB2120_MPP_ITC_IPC".RESET_FAULTS )
   END_RUNG wire#w1
   // the same network as SCL:
   #U02_TEMP_LOW_LIMIT_ALARM := ((#AUX_COOLING_SENSOR_U02_VALUES.COOLING_TEMP_SENSOR_ACTUAL_VALUE <= #AUX_COOLING_SENSOR_U02_VALUES.COOLING_TEMP_LOW_ALARM_HMI_VALUE) OR (#U02_TEMP_LOW_LIMIT_ALARM AND NOT "DB2120_MPP_ITC_IPC".RESET_FAULTS)) AND #O_BYTE_1.SECOND_FEEDBACK_FLOW_TEMP_SENSOR AND #IN_SERVICE;
END_REGION

REGION Network 47: UNIT 02 TEMPERATURE LOW LIMIT WARNING
   RUNG wire#powerrail
      { S7_Templates := "SrcType := Real" } LE_Contact(in1 := #AUX_COOLING_SENSOR_U02_VALUES.COOLING_TEMP_SENSOR_ACTUAL_VALUE, in2 := #AUX_COOLING_SENSOR_U02_VALUES.COOLING_TEMP_LOW_WARNING_HMI_VALUE)
      wire#w1
      Contact( #O_BYTE_1.SECOND_FEEDBACK_FLOW_TEMP_SENSOR )
      Contact( #IN_SERVICE )
      Coil( #U02_TEMP_LOW_LIMIT_WARNING )
   END_RUNG
   RUNG wire#powerrail
      Contact( #U02_TEMP_LOW_LIMIT_WARNING )
      I_Contact( "DB2120_MPP_ITC_IPC".RESET_FAULTS )
   END_RUNG wire#w1
   // the same network as SCL:
   #U02_TEMP_LOW_LIMIT_WARNING := ((#AUX_COOLING_SENSOR_U02_VALUES.COOLING_TEMP_SENSOR_ACTUAL_VALUE <= #AUX_COOLING_SENSOR_U02_VALUES.COOLING_TEMP_LOW_WARNING_HMI_VALUE) OR (#U02_TEMP_LOW_LIMIT_WARNING AND NOT "DB2120_MPP_ITC_IPC".RESET_FAULTS)) AND #O_BYTE_1.SECOND_FEEDBACK_FLOW_TEMP_SENSOR AND #IN_SERVICE;
END_REGION

REGION Network 48: UNIT 02 FLOW SETPOINT ALARM
   RUNG wire#powerrail
      Contact( #U02_FLOW_ACTUAL_RAW_VALUE.%X0 )
      wire#w1
      Contact( #O_BYTE_1.SECOND_FEEDBACK_FLOW_TEMP_SENSOR )
      Contact( #O_BYTE_1.U02_FLOW_SETPOINT_ALARM )
      Contact( #IN_SERVICE )
      Coil( #U02_FLOW_SETPOINT_ALARM )
   END_RUNG
   RUNG wire#powerrail
      Contact( #U02_FLOW_SETPOINT_ALARM )
      I_Contact( "DB2120_MPP_ITC_IPC".RESET_FAULTS )
   END_RUNG wire#w1
   // the same network as SCL:
   #U02_FLOW_SETPOINT_ALARM := (#U02_FLOW_ACTUAL_RAW_VALUE.%X0 OR (#U02_FLOW_SETPOINT_ALARM AND NOT "DB2120_MPP_ITC_IPC".RESET_FAULTS)) AND #O_BYTE_1.SECOND_FEEDBACK_FLOW_TEMP_SENSOR AND #O_BYTE_1.U02_FLOW_SETPOINT_ALARM AND #IN_SERVICE;
END_REGION

REGION Network 49: UNIT 02 TEMPERATURE SETPOINT ALARM
   RUNG wire#powerrail
      Contact( #U02_TEMP_ACTUAL_RAW_VALUE.%X0 )
      wire#w1
      Contact( #O_BYTE_1.SECOND_FEEDBACK_FLOW_TEMP_SENSOR )
      Contact( #O_BYTE_1.U02_TEMP_SETPOINT_ALARM )
      Contact( #IN_SERVICE )
      Coil( #U02_TEMP_SETPOINT_ALARM )
   END_RUNG
   RUNG wire#powerrail
      Contact( #U02_TEMP_SETPOINT_ALARM )
      I_Contact( "DB2120_MPP_ITC_IPC".RESET_FAULTS )
   END_RUNG wire#w1
   // the same network as SCL:
   #U02_TEMP_SETPOINT_ALARM := (#U02_TEMP_ACTUAL_RAW_VALUE.%X0 OR (#U02_TEMP_SETPOINT_ALARM AND NOT "DB2120_MPP_ITC_IPC".RESET_FAULTS)) AND #O_BYTE_1.SECOND_FEEDBACK_FLOW_TEMP_SENSOR AND #O_BYTE_1.U02_TEMP_SETPOINT_ALARM AND #IN_SERVICE;
END_REGION

REGION Network 50: STOP END OF CYCLE ALARMS
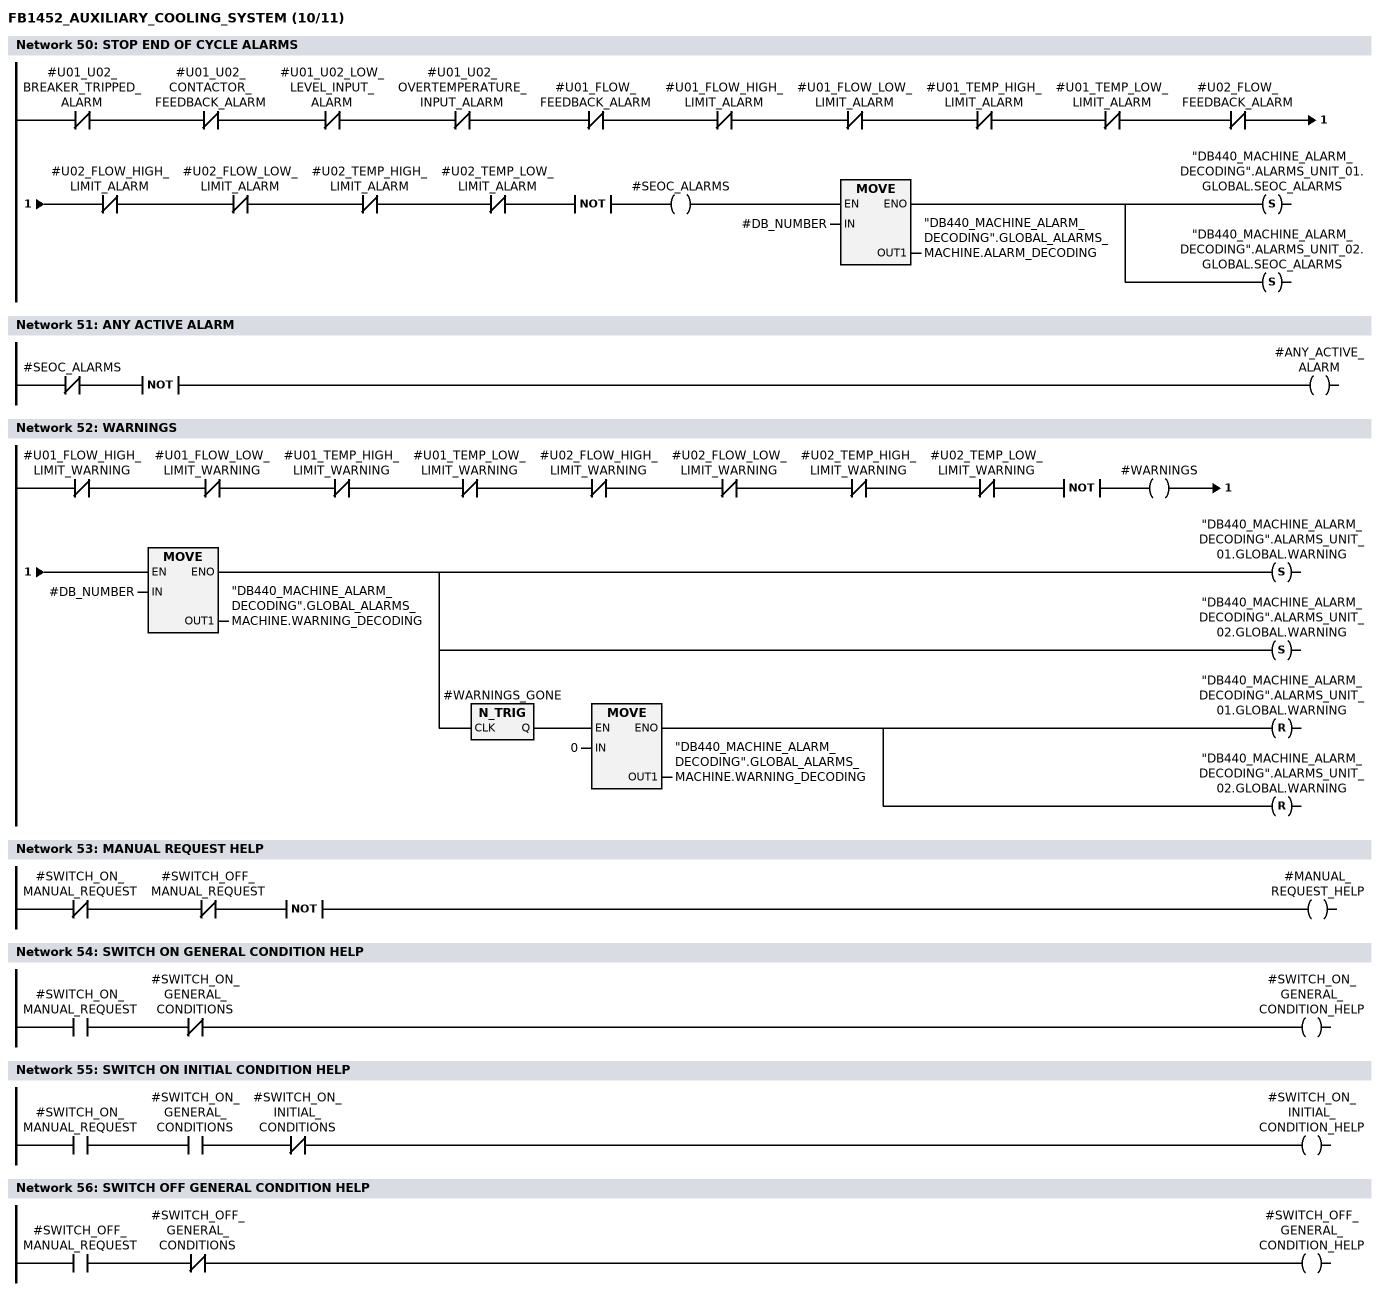
   RUNG wire#powerrail
      I_Contact( #U01_U02_BREAKER_TRIPPED_ALARM )
      I_Contact( #U01_U02_CONTACTOR_FEEDBACK_ALARM )
      I_Contact( #U01_U02_LOW_LEVEL_INPUT_ALARM )
      I_Contact( #U01_U02_OVERTEMPERATURE_INPUT_ALARM )
      I_Contact( #U01_FLOW_FEEDBACK_ALARM )
      I_Contact( #U01_FLOW_HIGH_LIMIT_ALARM )
      I_Contact( #U01_FLOW_LOW_LIMIT_ALARM )
      I_Contact( #U01_TEMP_HIGH_LIMIT_ALARM )
      I_Contact( #U01_TEMP_LOW_LIMIT_ALARM )
      I_Contact( #U02_FLOW_FEEDBACK_ALARM )
      I_Contact( #U02_FLOW_HIGH_LIMIT_ALARM )
      I_Contact( #U02_FLOW_LOW_LIMIT_ALARM )
      I_Contact( #U02_TEMP_HIGH_LIMIT_ALARM )
      I_Contact( #U02_TEMP_LOW_LIMIT_ALARM )
      Not()
      Coil( #SEOC_ALARMS )
      Move(in := #DB_NUMBER, out1 => "DB440_MACHINE_ALARM_DECODING".GLOBAL_ALARMS_MACHINE.ALARM_DECODING)
      wire#w1
      S_Coil( "DB440_MACHINE_ALARM_DECODING".ALARMS_UNIT_01.GLOBAL.SEOC_ALARMS )
   END_RUNG
   RUNG wire#w1
      S_Coil( "DB440_MACHINE_ALARM_DECODING".ALARMS_UNIT_02.GLOBAL.SEOC_ALARMS )
   END_RUNG
   // the same network as SCL:
   #SEOC_ALARMS := NOT (NOT #U01_U02_BREAKER_TRIPPED_ALARM AND NOT #U01_U02_CONTACTOR_FEEDBACK_ALARM AND NOT #U01_U02_LOW_LEVEL_INPUT_ALARM AND NOT #U01_U02_OVERTEMPERATURE_INPUT_ALARM AND NOT #U01_FLOW_FEEDBACK_ALARM AND NOT #U01_FLOW_HIGH_LIMIT_ALARM AND NOT #U01_FLOW_LOW_LIMIT_ALARM AND NOT #U01_TEMP_HIGH_LIMIT_ALARM AND NOT #U01_TEMP_LOW_LIMIT_ALARM AND NOT #U02_FLOW_FEEDBACK_ALARM AND NOT #U02_FLOW_HIGH_LIMIT_ALARM AND NOT #U02_FLOW_LOW_LIMIT_ALARM AND NOT #U02_TEMP_HIGH_LIMIT_ALARM AND NOT #U02_TEMP_LOW_LIMIT_ALARM);
   IF #SEOC_ALARMS THEN
       "DB440_MACHINE_ALARM_DECODING".GLOBAL_ALARMS_MACHINE.ALARM_DECODING := #DB_NUMBER;
       "DB440_MACHINE_ALARM_DECODING".ALARMS_UNIT_01.GLOBAL.SEOC_ALARMS := TRUE;
       "DB440_MACHINE_ALARM_DECODING".ALARMS_UNIT_02.GLOBAL.SEOC_ALARMS := TRUE;
   END_IF;
END_REGION

REGION Network 51: ANY ACTIVE ALARM
   RUNG wire#powerrail
      I_Contact( #SEOC_ALARMS )
      Not()
      Coil( #ANY_ACTIVE_ALARM )
   END_RUNG
   // the same network as SCL:
   #ANY_ACTIVE_ALARM := NOT (NOT #SEOC_ALARMS);
END_REGION

REGION Network 52: WARNINGS
   RUNG wire#powerrail
      I_Contact( #U01_FLOW_HIGH_LIMIT_WARNING )
      I_Contact( #U01_FLOW_LOW_LIMIT_WARNING )
      I_Contact( #U01_TEMP_HIGH_LIMIT_WARNING )
      I_Contact( #U01_TEMP_LOW_LIMIT_WARNING )
      I_Contact( #U02_FLOW_HIGH_LIMIT_WARNING )
      I_Contact( #U02_FLOW_LOW_LIMIT_WARNING )
      I_Contact( #U02_TEMP_HIGH_LIMIT_WARNING )
      I_Contact( #U02_TEMP_LOW_LIMIT_WARNING )
      Not()
      Coil( #WARNINGS )
      Move(in := #DB_NUMBER, out1 => "DB440_MACHINE_ALARM_DECODING".GLOBAL_ALARMS_MACHINE.WARNING_DECODING)
      wire#w1
      S_Coil( "DB440_MACHINE_ALARM_DECODING".ALARMS_UNIT_01.GLOBAL.WARNING )
   END_RUNG
   RUNG wire#w1
      S_Coil( "DB440_MACHINE_ALARM_DECODING".ALARMS_UNIT_02.GLOBAL.WARNING )
   END_RUNG
   RUNG wire#w1
      N_Trig( #WARNINGS_GONE )
      Move(in := 0, out1 => "DB440_MACHINE_ALARM_DECODING".GLOBAL_ALARMS_MACHINE.WARNING_DECODING)
      wire#w2
      R_Coil( "DB440_MACHINE_ALARM_DECODING".ALARMS_UNIT_01.GLOBAL.WARNING )
   END_RUNG
   RUNG wire#w2
      R_Coil( "DB440_MACHINE_ALARM_DECODING".ALARMS_UNIT_02.GLOBAL.WARNING )
   END_RUNG
   // the same network as SCL:
   #WARNINGS := NOT (NOT #U01_FLOW_HIGH_LIMIT_WARNING AND NOT #U01_FLOW_LOW_LIMIT_WARNING AND NOT #U01_TEMP_HIGH_LIMIT_WARNING AND NOT #U01_TEMP_LOW_LIMIT_WARNING AND NOT #U02_FLOW_HIGH_LIMIT_WARNING AND NOT #U02_FLOW_LOW_LIMIT_WARNING AND NOT #U02_TEMP_HIGH_LIMIT_WARNING AND NOT #U02_TEMP_LOW_LIMIT_WARNING);
   IF #WARNINGS THEN
       "DB440_MACHINE_ALARM_DECODING".GLOBAL_ALARMS_MACHINE.WARNING_DECODING := #DB_NUMBER;
       "DB440_MACHINE_ALARM_DECODING".ALARMS_UNIT_01.GLOBAL.WARNING := TRUE;
       "DB440_MACHINE_ALARM_DECODING".ALARMS_UNIT_02.GLOBAL.WARNING := TRUE;
   END_IF;
   #_w1 := NOT #WARNINGS AND #WARNINGS_GONE;   // falling edge
   #WARNINGS_GONE := #WARNINGS;
   IF #_w1 THEN
       "DB440_MACHINE_ALARM_DECODING".GLOBAL_ALARMS_MACHINE.WARNING_DECODING := 0;
       "DB440_MACHINE_ALARM_DECODING".ALARMS_UNIT_01.GLOBAL.WARNING := FALSE;
       "DB440_MACHINE_ALARM_DECODING".ALARMS_UNIT_02.GLOBAL.WARNING := FALSE;
   END_IF;
END_REGION

REGION Network 53: MANUAL REQUEST HELP
   RUNG wire#powerrail
      I_Contact( #SWITCH_ON_MANUAL_REQUEST )
      I_Contact( #SWITCH_OFF_MANUAL_REQUEST )
      Not()
      Coil( #MANUAL_REQUEST_HELP )
   END_RUNG
   // the same network as SCL:
   #MANUAL_REQUEST_HELP := NOT (NOT #SWITCH_ON_MANUAL_REQUEST AND NOT #SWITCH_OFF_MANUAL_REQUEST);
END_REGION

REGION Network 54: SWITCH ON GENERAL CONDITION HELP
   RUNG wire#powerrail
      Contact( #SWITCH_ON_MANUAL_REQUEST )
      I_Contact( #SWITCH_ON_GENERAL_CONDITIONS )
      Coil( #SWITCH_ON_GENERAL_CONDITION_HELP )
   END_RUNG
   // the same network as SCL:
   #SWITCH_ON_GENERAL_CONDITION_HELP := #SWITCH_ON_MANUAL_REQUEST AND NOT #SWITCH_ON_GENERAL_CONDITIONS;
END_REGION

REGION Network 55: SWITCH ON INITIAL CONDITION HELP
   RUNG wire#powerrail
      Contact( #SWITCH_ON_MANUAL_REQUEST )
      Contact( #SWITCH_ON_GENERAL_CONDITIONS )
      I_Contact( #SWITCH_ON_INITIAL_CONDITIONS )
      Coil( #SWITCH_ON_INITIAL_CONDITION_HELP )
   END_RUNG
   // the same network as SCL:
   #SWITCH_ON_INITIAL_CONDITION_HELP := #SWITCH_ON_MANUAL_REQUEST AND #SWITCH_ON_GENERAL_CONDITIONS AND NOT #SWITCH_ON_INITIAL_CONDITIONS;
END_REGION

REGION Network 56: SWITCH OFF GENERAL CONDITION HELP
   RUNG wire#powerrail
      Contact( #SWITCH_OFF_MANUAL_REQUEST )
      I_Contact( #SWITCH_OFF_GENERAL_CONDITIONS )
      Coil( #SWITCH_OFF_GENERAL_CONDITION_HELP )
   END_RUNG
   // the same network as SCL:
   #SWITCH_OFF_GENERAL_CONDITION_HELP := #SWITCH_OFF_MANUAL_REQUEST AND NOT #SWITCH_OFF_GENERAL_CONDITIONS;
END_REGION

REGION Network 57: SWITCH OFF INITIAL CONDITION HELP
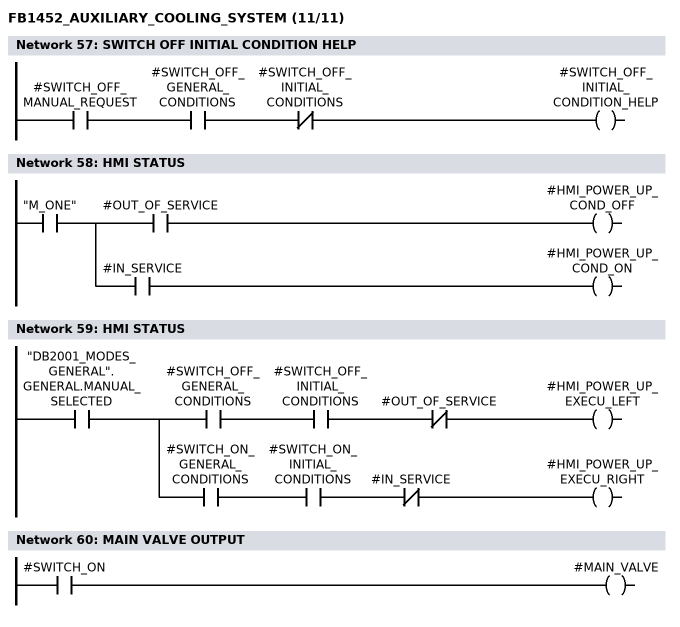
   RUNG wire#powerrail
      Contact( #SWITCH_OFF_MANUAL_REQUEST )
      Contact( #SWITCH_OFF_GENERAL_CONDITIONS )
      I_Contact( #SWITCH_OFF_INITIAL_CONDITIONS )
      Coil( #SWITCH_OFF_INITIAL_CONDITION_HELP )
   END_RUNG
   // the same network as SCL:
   #SWITCH_OFF_INITIAL_CONDITION_HELP := #SWITCH_OFF_MANUAL_REQUEST AND #SWITCH_OFF_GENERAL_CONDITIONS AND NOT #SWITCH_OFF_INITIAL_CONDITIONS;
END_REGION

REGION Network 58: HMI STATUS
   RUNG wire#powerrail
      Contact( "M_ONE" )
      wire#w1
      Contact( #OUT_OF_SERVICE )
      Coil( #HMI_POWER_UP_COND_OFF )
   END_RUNG
   RUNG wire#w1
      Contact( #IN_SERVICE )
      Coil( #HMI_POWER_UP_COND_ON )
   END_RUNG
   // the same network as SCL:
   #HMI_POWER_UP_COND_OFF := "M_ONE" AND #OUT_OF_SERVICE;
   #HMI_POWER_UP_COND_ON := "M_ONE" AND #IN_SERVICE;
END_REGION

REGION Network 59: HMI STATUS
   RUNG wire#powerrail
      Contact( "DB2001_MODES_GENERAL".GENERAL.MANUAL_SELECTED )
      wire#w1
      Contact( #SWITCH_OFF_GENERAL_CONDITIONS )
      Contact( #SWITCH_OFF_INITIAL_CONDITIONS )
      I_Contact( #OUT_OF_SERVICE )
      Coil( #HMI_POWER_UP_EXECU_LEFT )
   END_RUNG
   RUNG wire#w1
      Contact( #SWITCH_ON_GENERAL_CONDITIONS )
      Contact( #SWITCH_ON_INITIAL_CONDITIONS )
      I_Contact( #IN_SERVICE )
      Coil( #HMI_POWER_UP_EXECU_RIGHT )
   END_RUNG
   // the same network as SCL:
   #HMI_POWER_UP_EXECU_LEFT := "DB2001_MODES_GENERAL".GENERAL.MANUAL_SELECTED AND #SWITCH_OFF_GENERAL_CONDITIONS AND #SWITCH_OFF_INITIAL_CONDITIONS AND NOT #OUT_OF_SERVICE;
   #HMI_POWER_UP_EXECU_RIGHT := "DB2001_MODES_GENERAL".GENERAL.MANUAL_SELECTED AND #SWITCH_ON_GENERAL_CONDITIONS AND #SWITCH_ON_INITIAL_CONDITIONS AND NOT #IN_SERVICE;
END_REGION

REGION Network 60: MAIN VALVE OUTPUT
   RUNG wire#powerrail
      Contact( #SWITCH_ON )
      Coil( #MAIN_VALVE )
   END_RUNG
   // the same network as SCL:
   #MAIN_VALVE := #SWITCH_ON;
END_REGION
END_FUNCTION_BLOCK
